# B&R Automation Studio project 2SegDemo (part 2)

#### Cyclic.st
```iecst
PROGRAM _CYCLIC

	FOR i:= 0 TO gMainIf.Cfg.ShuttleCount - 1 DO
		IF NOT gShuttleIf[i].Cmd.Enable AND gShuttleIf[i].Sts.Active THEN
			shState[i] := SH_RESET;
		END_IF

		CASE shState[i] OF
			SH_OFF:  //******************************************************************************** Shuttle is in the off/idle state
				IF gShuttleIf[i].Cmd.Enable THEN
					shState[i] := SH_INIT;
				ELSE

				END_IF
			SH_INIT:  //******************************************************************************** Shuttle is in the initilization state
				//In this state we could make any checks on the current shuttle process perhaps in order to aide in recovery?

				shState[i] := SH_STARTUP;
			SH_STARTUP:  //******************************************************************************** Shuttle is in the startup state
				//In this state maybe we have triggered recovery and we're waiting for the autodrive to complete
				shState[i] := SH_IDLE;

			SH_IDLE:  //************************* ******************************************************* Shuttle is in the idle state
				shFbs[i].MovePlane.Controller := ADR(gMcAcp6DController);
				shFbs[i].MovePlane.ShuttleID := gShuttleIf[i].Cfg.ShuttleId;
				shFbs[i].MovePlane.Velocity := gProcessRecipe.General.Velocity;
				shFbs[i].MovePlane.Acceleration := gProcessRecipe.General.Accel;
				shFbs[i].MovePlane.EndVelocity := 0;
				shFbs[i].MovePlane.PositionX := gLoadStIf.Cfg.StationPos.X;
				shFbs[i].MovePlane.PositionY := gLoadStIf.Cfg.StationPos.Y;
				shFbs[i].MovePlane.Mode := mcACP6D_MOVE_ABSOLUTE;
				shFbs[i].MovePlane.Path := mcACP6D_PATH_Y_THEN_X;
				shFbs[i].MovePlane.Execute := TRUE;

				gShuttleIf[i].Sts.Active := TRUE;
				gShuttleIf[i].Sts.CurrentDestination := DEST_LOAD;

				shState[i] := SH_GO_TO_LOAD;

			SH_GO_TO_LOAD: //******************************************************************************** Shuttle is moving to the load station
				IF shFbs[i].MovePlane.Error THEN
					gShuttleIf[i].Sts.Error := TRUE;
					gShuttleIf[i].Sts.ErrorState := shState[i];

					logArgs[0] := ADR(i);
					logArgs[1] := ADR(shFbs[i].MovePlane.ErrorID);
					logError('ShCtrl','Sh%d had error %d moving to load',ADR(logArgs));

					shState[i] := SH_ERROR;
				ELSIF shFbs[i].MovePlane.Done AND (gLoadStIf.Par.ShuttleIdx = STATION_IS_EMPTY AND gLoadStIf.Sts.ReadyForNewShuttle)
					AND PositionValidation(ADR(gLoadStIf.Cfg.StationPos),ADR(gShuttleIf[i].Sts.ShuttleInfo.Position)) THEN
					gLoadStIf.Par.ShuttleIdx := i;
					gLoadStIf.Cmd.Process := TRUE;

					logArgs[0] := ADR(i);
					logDebug('ShCtrl','Sh%d arrived at Load',ADR(logArgs));

					shFbs[i].MovePlane.Execute := FALSE;
					shState[i] := SH_LOADING;
				END_IF
			SH_LOADING://******************************************************************************** Shuttle is at the load station
				IF gShuttleIf[i].Cmd.NextStep THEN
					gShuttleIf[i].Cmd.NextStep := FALSE;
					gLoadStIf.Cmd.Process := FALSE;

					gShuttleIf[i].Sts.LoopCounter := RandValueDINT(1,gProcessRecipe.General.St1St2Cycles);

					logArgs[0] := ADR(i);
					logDebug('ShCtrl','Sh%d Load complete',ADR(logArgs));

					shState[i] := SH_CHECK_RECIPE;
				END_IF
			SH_CHECK_RECIPE: //******************************************************************************** Shuttle is being checked for the recipe values
				IF gShuttleIf[i].Sts.LoopCounter <= 0 THEN
					shFbs[i].MovePlane.Controller := ADR(gMcAcp6DController);
					shFbs[i].MovePlane.ShuttleID := gShuttleIf[i].Cfg.ShuttleId;
					shFbs[i].MovePlane.Velocity := gProcessRecipe.General.Velocity;
					shFbs[i].MovePlane.Acceleration := gProcessRecipe.General.Accel;
					shFbs[i].MovePlane.EndVelocity := 0;

					shFbs[i].MovePlane.PositionX := gInspectIf.Cfg.StationPos.X;
					shFbs[i].MovePlane.PositionY := gInspectIf.Cfg.StationPos.Y;
					shFbs[i].MovePlane.Mode := mcACP6D_MOVE_ABSOLUTE;
					shFbs[i].MovePlane.Path := mcACP6D_PATH_X_THEN_Y;
					shFbs[i].MovePlane.Execute := TRUE;

					logArgs[0] := ADR(i);
					logDebug('ShCtrl','Sh%d sending to Inspect',ADR(logArgs));

					gShuttleIf[i].Sts.CurrentDestination := DEST_INSPECT;
					shState[i] := SH_GO_TO_INSPECT;
				ELSE

					shFbs[i].MovePlane.Controller := ADR(gMcAcp6DController);
					shFbs[i].MovePlane.ShuttleID := gShuttleIf[i].Cfg.ShuttleId;
					shFbs[i].MovePlane.Velocity := gProcessRecipe.General.Velocity;
					shFbs[i].MovePlane.Acceleration := gProcessRecipe.General.Accel;
					shFbs[i].MovePlane.EndVelocity := 0;

					shFbs[i].MovePlane.Mode := mcACP6D_MOVE_ABSOLUTE;
					shFbs[i].MovePlane.Path := mcACP6D_PATH_Y_THEN_X;
					shFbs[i].MovePlane.Execute := TRUE;

					logArgs[0] := ADR(i);
					logDebug('ShCtrl','Sh%d sending to Station 1',ADR(logArgs));

					gShuttleIf[i].Sts.CurrentDestination := DEST_PROCESS_1;
					shState[i] := SH_GO_TO_ST_1;
				END_IF

			SH_GO_TO_ST_1: //******************************************************************************** Shuttle is going to the #1 operating station
				IF shFbs[i].MovePlane.Error THEN
					gShuttleIf[i].Sts.Error := TRUE;
					gShuttleIf[i].Sts.ErrorState := shState[i];

					logArgs[0] := ADR(i);
					logArgs[1] := ADR(shFbs[i].MovePlane.ErrorID);
					logError('ShCtrl','Sh%d had error %d moving to Station 1',ADR(logArgs));

					shState[i] := SH_ERROR;
				ELSIF shFbs[i].MovePlane.Done AND (gProcessStIf[STATION_1].Par.ShuttleIdx = STATION_IS_EMPTY AND gProcessStIf[STATION_1].Sts.ReadyForNewShuttle)
					AND PositionValidation(ADR(gProcessStIf[STATION_1].Cfg.StationPos),ADR(gShuttleIf[i].Sts.ShuttleInfo.Position)) THEN
					gProcessStIf[STATION_1].Par.ShuttleIdx := i;
					gProcessStIf[STATION_1].Cmd.Process := TRUE;

					logArgs[0] := ADR(i);
					logDebug('ShCtrl','Sh%d arrived at Station 1',ADR(logArgs));

					shFbs[i].MovePlane.Execute := FALSE;
					shState[i] := SH_PREFORM_ST_1;
				END_IF
			SH_PREFORM_ST_1: //******************************************************************************** Shuttle is being operated on at station 1
				IF gShuttleIf[i].Cmd.NextStep THEN
					gShuttleIf[i].Cmd.NextStep := FALSE;

					shFbs[i].MovePlane.Controller := ADR(gMcAcp6DController);
					shFbs[i].MovePlane.ShuttleID := gShuttleIf[i].Cfg.ShuttleId;
					shFbs[i].MovePlane.Velocity := gProcessRecipe.General.Velocity;
					shFbs[i].MovePlane.Acceleration := gProcessRecipe.General.Accel;
					shFbs[i].MovePlane.EndVelocity := 0;
					shFbs[i].MovePlane.PositionX := gProcessStIf[STATION_2].Cfg.StationPos.X;
					shFbs[i].MovePlane.PositionY := gProcessStIf[STATION_2].Cfg.StationPos.Y;
					shFbs[i].MovePlane.Mode := mcACP6D_MOVE_ABSOLUTE;
					shFbs[i].MovePlane.Path := mcACP6D_PATH_Y_THEN_X;
					shFbs[i].MovePlane.Execute := TRUE;

					logArgs[0] := ADR(i);
					logDebug('ShCtrl','Sh%d sent to Station 2',ADR(logArgs));

					gShuttleIf[i].Sts.CurrentDestination := DEST_PROCESS_2;
					shState[i] := SH_GO_TO_ST_2;
				END_IF
			SH_GO_TO_ST_2: //******************************************************************************** Shuttle is going to the #2 operating station
				IF shFbs[i].MovePlane.Error THEN
					gShuttleIf[i].Sts.Error := TRUE;
					gShuttleIf[i].Sts.ErrorState := shState[i];

					logArgs[0] := ADR(i);
					logArgs[1] := ADR(shFbs[i].MovePlane.ErrorID);
					logError('ShCtrl','Sh%d had error %d moving to Station 2',ADR(logArgs));

					shState[i] := SH_ERROR;
				ELSIF shFbs[i].MovePlane.Done AND (gProcessStIf[STATION_2].Par.ShuttleIdx = STATION_IS_EMPTY AND gProcessStIf[STATION_2].Sts.ReadyForNewShuttle)
					AND PositionValidation(ADR(gProcessStIf[STATION_2].Cfg.StationPos),ADR(gShuttleIf[i].Sts.ShuttleInfo.Position)) THEN
					gProcessStIf[STATION_2].Par.ShuttleIdx := i;
					gProcessStIf[STATION_2].Cmd.Process := TRUE;

					logArgs[0] := ADR(i);
					logDebug('ShCtrl','Sh%d arrived at Station 2',ADR(logArgs));

					shFbs[i].MovePlane.Execute := FALSE;
					shState[i] := SH_PREFORM_ST_2;
				END_IF
			SH_PREFORM_ST_2: //******************************************************************************** Shuttle is being operated on at station 2
				IF gShuttleIf[i].Cmd.NextStep THEN
					gShuttleIf[i].Cmd.NextStep := FALSE;

					logArgs[0] := ADR(i);
					logDebug('ShCtrl','Sh%d sent to inspection',ADR(logArgs));

					shState[i] := SH_CHECK_RECIPE;
				END_IF
			SH_GO_TO_INSPECT: //******************************************************************************** Shuttle is going to the inspection station
				IF shFbs[i].MovePlane.Error THEN
					gShuttleIf[i].Sts.Error := TRUE;
					gShuttleIf[i].Sts.ErrorState := shState[i];

					logArgs[0] := ADR(i);
					logArgs[1] := ADR(shFbs[i].MovePlane.ErrorID);
					logError('ShCtrl','Sh%d had error %d moving to inspection',ADR(logArgs));

					shState[i] := SH_ERROR;
				ELSIF shFbs[i].MovePlane.Done AND (gInspectIf.Par.ShuttleIdx = STATION_IS_EMPTY AND gInspectIf.Sts.ReadyForNewShuttle)
						AND PositionValidation(ADR(gInspectIf.Cfg.StationPos),ADR(gShuttleIf[i].Sts.ShuttleInfo.Position)) THEN
					gInspectIf.Par.ShuttleIdx := i;
					gInspectIf.Cmd.Process := TRUE;

					logArgs[0] := ADR(i);
					logDebug('ShCtrl','Sh%d arrived at inspection',ADR(logArgs));

					shFbs[i].MovePlane.Execute := FALSE;
					shState[i] := SH_INSPECT;
				END_IF
			SH_INSPECT: //******************************************************************************** Shuttle is being operated on at the inspection station
				IF gShuttleIf[i].Cmd.NextStep THEN
					gShuttleIf[i].Cmd.NextStep := FALSE;

					shFbs[i].MovePlane.Controller := ADR(gMcAcp6DController);
					shFbs[i].MovePlane.ShuttleID := gShuttleIf[i].Cfg.ShuttleId;
					shFbs[i].MovePlane.Velocity := gProcessRecipe.General.Velocity;
					shFbs[i].MovePlane.Acceleration := gProcessRecipe.General.Accel;
					shFbs[i].MovePlane.EndVelocity := 0;
					shFbs[i].MovePlane.PositionX := gUnloadStIf.Cfg.StationPos.X;
					shFbs[i].MovePlane.PositionY := gUnloadStIf.Cfg.StationPos.Y;
					shFbs[i].MovePlane.Mode := mcACP6D_MOVE_ABSOLUTE;
					shFbs[i].MovePlane.Path := mcACP6D_PATH_Y_THEN_X;
					shFbs[i].MovePlane.Execute := TRUE;

					logArgs[0] := ADR(i);
					logDebug('ShCtrl','Sh%d sent to unload',ADR(logArgs));

					gShuttleIf[i].Sts.CurrentDestination := DEST_UNLOAD;
					shState[i] := SH_GO_TO_UNLOAD;
				END_IF
			SH_GO_TO_UNLOAD: //******************************************************************************** Shuttle is going to the unload station
				IF shFbs[i].MovePlane.Error THEN
					gShuttleIf[i].Sts.Error := TRUE;
					gShuttleIf[i].Sts.ErrorState := shState[i];

					logArgs[0] := ADR(i);
					logArgs[1] := ADR(shFbs[i].MovePlane.ErrorID);
					logError('ShCtrl','Sh%d had error %d moving to unload',ADR(logArgs));

					shState[i] := SH_ERROR;
				ELSIF shFbs[i].MovePlane.Done AND (gUnloadStIf.Par.ShuttleIdx = STATION_IS_EMPTY AND gUnloadStIf.Sts.ReadyForNewShuttle)
						AND PositionValidation(ADR(gUnloadStIf.Cfg.StationPos),ADR(gShuttleIf[i].Sts.ShuttleInfo.Position)) THEN
					gUnloadStIf.Par.ShuttleIdx := i;
					gUnloadStIf.Cmd.Process := TRUE;

					logArgs[0] := ADR(i);
					logDebug('ShCtrl','Sh%d arrived at unload',ADR(logArgs));

					shFbs[i].MovePlane.Execute := FALSE;
					shState[i] := SH_UNLOAD;
				END_IF
			SH_UNLOAD: //******************************************************************************** Shuttle is being operated on at the unload station
				IF gShuttleIf[i].Cmd.NextStep THEN
					gShuttleIf[i].Cmd.NextStep := FALSE;

					shFbs[i].MovePlane.Controller := ADR(gMcAcp6DController);
					shFbs[i].MovePlane.ShuttleID := gShuttleIf[i].Cfg.ShuttleId;
					//shFbs[i].MovePlane.Velocity := gProcessRecipe.General.Velocity;
					shFbs[i].MovePlane.Velocity := 0.5;
					shFbs[i].MovePlane.Acceleration := gProcessRecipe.General.Accel;
					shFbs[i].MovePlane.EndVelocity := 0;
					shFbs[i].MovePlane.PositionX := gLoadStIf.Cfg.StationPos.X;
					shFbs[i].MovePlane.PositionY := gLoadStIf.Cfg.StationPos.Y;
					shFbs[i].MovePlane.Mode := mcACP6D_MOVE_ABSOLUTE;
					shFbs[i].MovePlane.Path := mcACP6D_PATH_Y_THEN_X;
					shFbs[i].MovePlane.Execute := TRUE;

					logArgs[0] := ADR(i);
					logDebug('ShCtrl','Sh%d sent to load',ADR(logArgs));
					gShuttleIf[i].Cmd.ResetProductInfo := TRUE;

					gShuttleIf[i].Sts.CurrentDestination := DEST_LOAD;
					shState[i] := SH_GO_TO_LOAD;
				END_IF
			SH_STOPPING: //******************************************************************************** Shuttle is in the stopping state
				IF shFbs[i].Stop.Error THEN
					shState[i] := SH_ERROR;
				ELSIF gShuttleIf[i].Sts.ShuttleInfo.State.Valid AND
						(gShuttleIf[i].Sts.ShuttleInfo.State.Value = mcACP6D_SH_STATE_IDLING OR gShuttleIf[i].Sts.ShuttleInfo.State.Value = mcACP6D_SH_STATE_DISABLED) THEN
					gShuttleIf[i].Cmd.NextStep := FALSE;

					shFbs[i].Stop.Execute := FALSE;
					shFbs[i].MovePlane.Execute := FALSE;
					shFbs[i].ShRunMacroFb.Execute := FALSE;

					shState[i] := SH_RESET;
				END_IF

			SH_ERROR: //******************************************************************************** Shuttle is in the error state
				IF gShuttleIf[i].Cmd.Reset THEN
					shState[i] := SH_RESET;
				END_IF
			SH_RESET: //******************************************************************************** Reset all shuttle values
				gShuttleIf[i].Cmd.ResetProductInfo := TRUE;
				gShuttleIf[i].Cmd.Reset := FALSE;
				gShuttleIf[i].Cmd.NextStep := FALSE;
				gShuttleIf[i].Cmd.RunProcessDemo := FALSE;

				gShuttleIf[i].Sts.Active := FALSE;

				shFbs[i].MovePlane.Execute := FALSE;
				shFbs[i].ShRunMacroFb.Execute := FALSE;
				shFbs[i].Stop.Execute := FALSE;

				shState[i] := SH_OFF;
		END_CASE;

		shFbs[i].Stop();
		shFbs[i].MovePlane();

		IF gShuttleIf[i].Cmd.ResetProductInfo THEN
			gShuttleIf[i].Sts.Error := FALSE;
			gShuttleIf[i].Sts.ErrorState := 0;
			gShuttleIf[i].Cmd.ResetProductInfo := FALSE;
			gShuttleIf[i].Sts.LoopCounter := 0;
			gShuttleIf[i].Sts.ProductState := PROD_EMPTY;
			brsmemset(ADR(gShuttleIf[i].Sts.ProdFill),0,SIZEOF(gShuttleIf[i].Sts.ProdFill));
		END_IF

	END_FOR;

	pDebugIf ACCESS ADR(gShuttleIf[debugIdx]);
	pDebugState ACCESS ADR(shState[debugIdx]);
	pDebugFbs ACCESS ADR(shFbs[debugIdx]);

END_PROGRAM
```

#### Init.st
```iecst
PROGRAM _INIT

	FOR i:=0 TO gMainIf.Cfg.ShuttleCount-1 DO
		gShuttleIf[i].Par.X := 0.06;
		gShuttleIf[i].Par.Y := 0.06 * (i + 1) + 0.06*i;
		gShuttleIf[i].Par.Accel := 10;
		gShuttleIf[i].Par.Vel := 0.5;
		gShuttleIf[i].Par.EndVel := 0;
	END_FOR;
	gProcessRecipe.General.Velocity := 1;
	gProcessRecipe.General.Accel := 10;
END_PROGRAM
```

### Program Logical/Source/ShuttleCtrl/Recovery (IEC)

#### Types.typ
```iecst
TYPE
	RecoveryFbs : 	STRUCT
		AsyncMoveFb : MC_BR_MoveInPlaneAsync_Acp6D;
		ShStopFb : MC_BR_Stop_Acp6D;
		DelayFb : TON;
	END_STRUCT;
	RecoveryStateEnum :
		(
		RECOVER_IDLE, (*Recovery is in an idle state*)
		RECOVER_INIT, (*Initalize recovery state*)
		RECOVER_AUTODRIVE, (*Preform autodrive movement for recovery*)
		RECOVER_STOP,
		RECOVER_DONE, (*Recovery has been completed*)
		RECOVER_ERROR (*Recovery had an error*)
		);
END_TYPE
```

#### Variables.var
```iecst
VAR
	state : RecoveryStateEnum;
	RecoverFbs : RecoveryFbs;
	i : USINT;
END_VAR
```

#### Cyclic.st
```iecst
PROGRAM _CYCLIC

	(*
	Shuttle reocvery
		Move all shuttles to autodrive positions
		Wait for autodrive to be finished
		loop through each shuttle
			if that shuttle's group is current
				it is not recovered,
					groupRecovered=false
					Evaluate each shuttle's position
					Send it to the unload position and set the "Next step cmd" to be true
				else
					onwards, do nothing

	*)

	CASE state OF
		RECOVER_IDLE:   //******************************************************************************** Recovery is in an idle state*)
			IF g6DRecoveryIf.Cmd.Recover THEN
				g6DRecoveryIf.Sts.Recovering := TRUE;
				state := RECOVER_INIT;
			END_IF
		RECOVER_INIT:   //******************************************************************************** Initalize recovery state*)
			RecoverFbs.AsyncMoveFb.Controller := ADR(gMcAcp6DController);
			RecoverFbs.AsyncMoveFb.NumberOfShuttles := gMainIf.Cfg.ShuttleCount;
			RecoverFbs.AsyncMoveFb.Velocity := g6DRecoveryIf.Par.Vel;
			RecoverFbs.AsyncMoveFb.Acceleration := g6DRecoveryIf.Par.Accel;
			FOR i:=0 TO gMainIf.Cfg.ShuttleCount - 1 DO
				RecoverFbs.AsyncMoveFb.PositionX[i] := g6DRecoveryIf.Par.AutoDrivePositions[i].X;
				RecoverFbs.AsyncMoveFb.PositionY[i] := g6DRecoveryIf.Par.AutoDrivePositions[i].Y;
				RecoverFbs.AsyncMoveFb.ShuttleID[i] := gShuttleIf[g6DRecoveryIf.Par.AutoDrivePositions[i].ShIdx].Cfg.ShuttleId;
				IF RecoverFbs.AsyncMoveFb.ShuttleID[i] = 0 THEN// Invalid shuttle id here
					g6DRecoveryIf.Sts.Error := TRUE;
				END_IF
			END_FOR;
			IF NOT g6DRecoveryIf.Sts.Error THEN
				RecoverFbs.AsyncMoveFb.Execute := TRUE;
				state := RECOVER_AUTODRIVE;
			ELSE
				state := RECOVER_ERROR;
			END_IF

		RECOVER_AUTODRIVE:   //******************************************************************************** Preform autodrive movement for recovery*)
			IF RecoverFbs.AsyncMoveFb.Error AND RecoverFbs.AsyncMoveFb.ErrorID = mcACP6D_ERR_WRONG_SH_STATE THEN
				RecoverFbs.AsyncMoveFb.Execute := FALSE;

				RecoverFbs.DelayFb.IN := TRUE;
				RecoverFbs.DelayFb.PT := T#5s;

				RecoverFbs.ShStopFb.Controller := ADR(gMcAcp6DController);
				RecoverFbs.ShStopFb.ShuttleID := 0;
				RecoverFbs.ShStopFb.Execute := TRUE;

				state := RECOVER_STOP;
			ELSIF RecoverFbs.AsyncMoveFb.Error THEN
				g6DRecoveryIf.Sts.Error := TRUE;
				state := RECOVER_ERROR;
			ELSIF RecoverFbs.AsyncMoveFb.Done THEN
				g6DRecoveryIf.Sts.ReadyToStartProc := TRUE;
				RecoverFbs.AsyncMoveFb.Execute := FALSE;

				state := RECOVER_DONE;
			END_IF
		RECOVER_STOP:  //******************************************************************************** Stop All shuttles
			IF RecoverFbs.ShStopFb.Error THEN
				g6DRecoveryIf.Sts.Error := TRUE;
				state := RECOVER_ERROR;
			ELSIF RecoverFbs.ShStopFb.Done AND RecoverFbs.DelayFb.Q THEN
				RecoverFbs.DelayFb.IN := FALSE;
				RecoverFbs.ShStopFb.Execute := FALSE;

				RecoverFbs.AsyncMoveFb.Execute := TRUE;

				state := RECOVER_AUTODRIVE;
			END_IF
		RECOVER_DONE:   //******************************************************************************** Recovery has been completed*)
			IF NOT g6DRecoveryIf.Cmd.Recover THEN
				g6DRecoveryIf.Cmd.Reset := FALSE;
				RecoverFbs.DelayFb.IN := FALSE;
				g6DRecoveryIf.Sts.Done := FALSE;
				g6DRecoveryIf.Sts.ReadyToStartProc := FALSE;
				g6DRecoveryIf.Sts.Recovering := FALSE;
				g6DRecoveryIf.Sts.ShuttlesRecovered := FALSE;
				g6DRecoveryIf.Sts.Error := FALSE;

				RecoverFbs.AsyncMoveFb.Execute := FALSE;
				state := RECOVER_IDLE;
			END_IF
		RECOVER_ERROR:   //******************************************************************************** Recovery had an error*)
			IF g6DRecoveryIf.Cmd.Reset THEN
				RecoverFbs.DelayFb.IN := FALSE;
				g6DRecoveryIf.Cmd.Reset := FALSE;
				g6DRecoveryIf.Cmd.Recover := FALSE;

				g6DRecoveryIf.Sts.Done := FALSE;
				g6DRecoveryIf.Sts.ReadyToStartProc := FALSE;
				g6DRecoveryIf.Sts.Recovering := FALSE;
				g6DRecoveryIf.Sts.ShuttlesRecovered := FALSE;
				g6DRecoveryIf.Sts.Error := FALSE;

				RecoverFbs.AsyncMoveFb.Execute := FALSE;
				RecoverFbs.ShStopFb.Execute := FALSE;
				state := RECOVER_IDLE;
			END_IF
	END_CASE;
	RecoverFbs.AsyncMoveFb();
	RecoverFbs.ShStopFb();
	RecoverFbs.DelayFb();
END_PROGRAM
```

#### Init.st
```iecst
PROGRAM _INIT
	g6DRecoveryIf.Par.Vel := 1;
	g6DRecoveryIf.Par.Accel := 10;

	//************************************************************************* Shuttle 1
	g6DRecoveryIf.Par.AutoDrivePositions[0].ShIdx := 0;
	g6DRecoveryIf.Par.AutoDrivePositions[0].X := 0.42;
	g6DRecoveryIf.Par.AutoDrivePositions[0].Y := 0.18;
	//************************************************************************* Shuttle 2
	g6DRecoveryIf.Par.AutoDrivePositions[1].ShIdx := 1;
	g6DRecoveryIf.Par.AutoDrivePositions[1].X := 0.30;
	g6DRecoveryIf.Par.AutoDrivePositions[1].Y := 0.18;
	//************************************************************************* Shuttle 3
	g6DRecoveryIf.Par.AutoDrivePositions[2].ShIdx := 2;
	g6DRecoveryIf.Par.AutoDrivePositions[2].X := 0.42;
	g6DRecoveryIf.Par.AutoDrivePositions[2].Y := 0.30;
	//************************************************************************* Shuttle 4
	g6DRecoveryIf.Par.AutoDrivePositions[3].ShIdx := 3;
	g6DRecoveryIf.Par.AutoDrivePositions[3].X := 0.30;
	g6DRecoveryIf.Par.AutoDrivePositions[3].Y := 0.30;
	//************************************************************************* Shuttle 5
	g6DRecoveryIf.Par.AutoDrivePositions[4].ShIdx := 4;
	g6DRecoveryIf.Par.AutoDrivePositions[4].X := 0.42;
	g6DRecoveryIf.Par.AutoDrivePositions[4].Y := 0.42;
	//************************************************************************* Shuttle 6
	g6DRecoveryIf.Par.AutoDrivePositions[5].ShIdx := 5;
	g6DRecoveryIf.Par.AutoDrivePositions[5].X := 0.30;
	g6DRecoveryIf.Par.AutoDrivePositions[5].Y := 0.42;
	//************************************************************************* Shuttle 7
	g6DRecoveryIf.Par.AutoDrivePositions[6].ShIdx := 6;
	g6DRecoveryIf.Par.AutoDrivePositions[6].X := 0.42;
	g6DRecoveryIf.Par.AutoDrivePositions[6].Y := 0.54;
	//************************************************************************* Shuttle 8
	g6DRecoveryIf.Par.AutoDrivePositions[7].ShIdx := 7;
	g6DRecoveryIf.Par.AutoDrivePositions[7].X := 0.30;
	g6DRecoveryIf.Par.AutoDrivePositions[7].Y := 0.54;

END_PROGRAM
```

### Program Logical/Source/ShuttleCtrl/ProcessDemoCtrl (IEC) - Control the process demo

#### Types.typ
```iecst
TYPE
	ProcessDemoStateEnum :
		(
		PROCESS_IDLE,
		PROCESS_ROUTING,
		PROCESS_STARTUP,
		PROCESS_RUN_DEMO,
		PROCESS_STOPPING_STATIONS,
		PROCESS_STOPPING,
		PROCESS_UNLOAD_PROGRAM,
		PROCESS_ERROR,
		PROCESS_RESET
		);
	ProcessDemoFbsTyp : 	STRUCT
		Stop6DFb : MC_BR_Stop_Acp6D;
		MoveProgramFb : MC_BR_MoveProgram;
		StopRobotFb : MC_GroupStop;
		UnloadProgramFb : MC_BR_UnloadProgram;
	END_STRUCT;
END_TYPE
```

#### Variables.var
```iecst
VAR
	state : ProcessDemoStateEnum;
	Fbs : ProcessDemoFbsTyp;
	i : USINT;
END_VAR
```

#### Cyclic.st
```iecst
(* This task control the demo routine for the process demo
	The robot and the 6D are expected to be powered on, homed and not in any error states before starting this demo

	Recovery
	Robot Setup
	Enable Stations
	Run Demo
	Error
	Stopping
	Reset
*)

PROGRAM _CYCLIC
	CASE state OF
		PROCESS_IDLE:  //******************************************************************************** Idle Wait State
			IF gProcessPickPlaceIf.Cmd.RunDemo THEN
				g6DRecoveryIf.Cmd.Recover := TRUE;

				state := PROCESS_ROUTING;
			ELSIF gProcessPickPlaceIf.Cmd.Reset THEN
				state := PROCESS_RESET;
			END_IF
		PROCESS_ROUTING:  //******************************************************************************** Running the routing demo
			IF g6DRecoveryIf.Sts.Error THEN
				gProcessPickPlaceIf.Sts.Error := TRUE;
				state := PROCESS_ERROR;
			ELSIF (g6DRecoveryIf.Sts.ReadyToStartProc) THEN
				g6DRecoveryIf.Cmd.Recover := FALSE;

				gLoadStIf.Cmd.Enable := TRUE;
				//gUnloadStIf.Cmd.Enable := TRUE; The Load station will enable the Unload station in order to complete the Load process first
				gProcessStIf[STATION_1].Cmd.Enable := TRUE;
				gProcessStIf[STATION_2].Cmd.Enable := TRUE;
				gInspectIf.Cmd.Enable := TRUE;

				Fbs.MoveProgramFb.AxesGroup := ADR(g3AxDeltaA);
				Fbs.MoveProgramFb.Name := 'ProcessDemo.gcode';
				Fbs.MoveProgramFb.Execute := TRUE;

				state := PROCESS_STARTUP;
			END_IF
		PROCESS_STARTUP:  //******************************************************************************** Starting up the demos state
			IF gLoadStIf.Sts.Error OR
					gInspectIf.Sts.Error OR
					gProcessStIf[STATION_1].Sts.Error OR
					gProcessStIf[STATION_2].Sts.Error OR
					Fbs.MoveProgramFb.Error THEN
				gProcessPickPlaceIf.Sts.Error := TRUE;
				state := PROCESS_ERROR;
			ELSIF (gLoadStIf.Sts.Enabled AND
					//gUnloadStIf.Sts.Enabled AND The load station enables the unload station once the startup process has completed
					gInspectIf.Cmd.Enable AND
					gProcessStIf[STATION_1].Sts.Enabled AND
					gProcessStIf[STATION_2].Sts.Enabled OR NOT gMainIf.Cfg.Enable6D)
					AND
					Fbs.MoveProgramFb.Phase = mcPRGPH_REAL_RUN THEN

				CmdShEnable(TRUE, ADR(gShuttleIf),gMainIf.Cfg.ShuttleCount);

				gProcessPickPlaceIf.Sts.DemoRunning := TRUE;

				state := PROCESS_RUN_DEMO;

			END_IF
		PROCESS_RUN_DEMO:  //******************************************************************************** Running the process demo
			IF Fbs.MoveProgramFb.Error OR
					gLoadStIf.Sts.Error OR
					gUnloadStIf.Sts.Error OR
					gProcessStIf[STATION_1].Sts.Error OR
					gProcessStIf[STATION_2].Sts.Error OR
					gInspectIf.Sts.Error THEN
				state := PROCESS_ERROR;
			ELSIF NOT gProcessPickPlaceIf.Cmd.RunDemo THEN
				gLoadStIf.Cmd.Enable := FALSE;
				gUnloadStIf.Cmd.Enable := FALSE;
				gProcessStIf[STATION_1].Cmd.Enable := FALSE;
				gProcessStIf[STATION_2].Cmd.Enable := FALSE;
				gInspectIf.Cmd.Enable := FALSE;

				state := PROCESS_STOPPING_STATIONS;
			END_IF
		PROCESS_STOPPING_STATIONS:  //******************************************************************************** Stopping the Stations
			gLoadStIf.Cmd.Enable := FALSE;
			gUnloadStIf.Cmd.Enable := FALSE;
			gProcessStIf[STATION_1].Cmd.Enable := FALSE;
			gProcessStIf[STATION_2].Cmd.Enable := FALSE;
			gInspectIf.Cmd.Enable := FALSE;
			IF (NOT gLoadStIf.Sts.Enabled AND
					//gUnloadStIf.Sts.Enabled AND The load station enables the unload station once the startup process has completed
					NOT gInspectIf.Cmd.Enable AND
					NOT gProcessStIf[STATION_1].Sts.Enabled AND
					NOT gProcessStIf[STATION_2].Sts.Enabled AND NOT gUnloadStIf.Sts.Enabled) AND Fbs.MoveProgramFb.Done
					THEN

				Fbs.StopRobotFb.AxesGroup := ADR(g3AxDeltaA);
				Fbs.StopRobotFb.Execute := TRUE;

				Fbs.Stop6DFb.Controller := ADR(gMcAcp6DController);
				Fbs.Stop6DFb.ShuttleID := 0;
				Fbs.Stop6DFb.Execute := TRUE;

				state := PROCESS_STOPPING;
			END_IF
		PROCESS_STOPPING:  //******************************************************************************** Stopping the demo
			IF Fbs.Stop6DFb.Error OR Fbs.StopRobotFb.Error THEN
				gProcessPickPlaceIf.Sts.Error := TRUE;

				state := PROCESS_ERROR;
			ELSIF Fbs.Stop6DFb.Done AND Fbs.StopRobotFb.Done THEN
				Fbs.StopRobotFb.Execute := FALSE;
				Fbs.Stop6DFb.Execute := FALSE;

				gProcessPickPlaceIf.Sts.DemoRunning := FALSE;

				FOR i:=0 TO gMainIf.Cfg.ShuttleCount - 1 DO
					gShuttleIf[i].Cmd.Enable := FALSE;
					gShuttleIf[i].Sts.Recovered := FALSE;
				END_FOR;

				Fbs.UnloadProgramFb.AxesGroup := ADR(g3AxDeltaA);
				Fbs.UnloadProgramFb.Execute := TRUE;
				Fbs.UnloadProgramFb.Mode := mcUNLOADPRG_ALL;

				state := PROCESS_UNLOAD_PROGRAM;
			END_IF
		PROCESS_UNLOAD_PROGRAM:   //******************************************************************************** Unloading the program
			IF Fbs.UnloadProgramFb.Error THEN
				gProcessPickPlaceIf.Sts.Error := TRUE;

				state := PROCESS_ERROR;
			ELSIF Fbs.UnloadProgramFb.Done THEN
				Fbs.UnloadProgramFb.Execute := FALSE;

				state := PROCESS_RESET;
			END_IF

		PROCESS_ERROR:  //******************************************************************************** Demo in error state
			IF gProcessPickPlaceIf.Cmd.Reset THEN
				gLoadStIf.Cmd.Reset := TRUE;
				gUnloadStIf.Cmd.Reset:= TRUE;
				gProcessStIf[STATION_1].Cmd.Reset := TRUE;
				gProcessStIf[STATION_2].Cmd.Reset := TRUE;
				gInspectIf.Cmd.Reset := TRUE;

				Fbs.Stop6DFb.Controller := ADR(gMcAcp6DController);
				Fbs.Stop6DFb.ShuttleID := 0;
				Fbs.Stop6DFb.Execute := TRUE;

				FOR i:= 0 TO gMainIf.Cfg.ShuttleCount - 1 DO
					gShuttleIf[i].Cmd.Enable := FALSE;
					gShuttleIf[i].Cmd.Reset := TRUE;
				END_FOR;
				state := PROCESS_RESET;
			END_IF
		PROCESS_RESET:  //******************************************************************************** Resetting the demo state
			Fbs.Stop6DFb.Execute := FALSE;
			Fbs.MoveProgramFb.Execute := FALSE;
			Fbs.StopRobotFb.Execute := FALSE;
			Fbs.UnloadProgramFb.Execute := FALSE;

			gDelta.Cmd.ErrorReset := gDelta.Status.Error;

			g6DRecoveryIf.Cmd.Reset := g6DRecoveryIf.Sts.Error;

			gLoadStIf.Cmd.Enable := FALSE;
			gUnloadStIf.Cmd.Enable := FALSE;
			gProcessStIf[STATION_1].Cmd.Enable := FALSE;
			gProcessStIf[STATION_2].Cmd.Enable := FALSE;
			gInspectIf.Cmd.Enable := FALSE;

			gProcessPickPlaceIf.Cmd.PickLoad := FALSE;
			gProcessPickPlaceIf.Cmd.PickUnload := FALSE;
			gProcessPickPlaceIf.Cmd.RunDemo := FALSE;
			gProcessPickPlaceIf.Cmd.GetLoadPart := FALSE;

			gProcessPickPlaceIf.Sts.Error := FALSE;
			gProcessPickPlaceIf.Sts.DemoRunning := FALSE;
			gProcessPickPlaceIf.Sts.FinishedProductPresent := FALSE;
			gProcessPickPlaceIf.Sts.ReadyForLoad := FALSE;
			gProcessPickPlaceIf.Sts.ReadyForUnload := FALSE;
			gProcessPickPlaceIf.Sts.StartupComplete := FALSE;
			gProcessPickPlaceIf.Sts.Sync := FALSE;
			gProcessPickPlaceIf.Sts.UnfinishedProductPresent := FALSE;
			gProcessPickPlaceIf.Cmd.Reset := FALSE;
			gProcessPickPlaceIf.Sts.Place := FALSE;

			state := PROCESS_IDLE;
	END_CASE;

	Fbs.Stop6DFb();
	Fbs.MoveProgramFb();
	Fbs.UnloadProgramFb();
	Fbs.StopRobotFb();
END_PROGRAM
```

#### Init.st
```iecst
PROGRAM _INIT
	gDanceDemoIf.Par.DemoTime := T#30s;

END_PROGRAM
```

### DemoGlobalVariables.var
```iecst
VAR
	gSyncConoyDemoIf : IndvDanceDemoIfTyp;
	gDofDemoIf : IndvDanceDemoIfTyp;
	gRoutingDemoIf : IndvDanceDemoIfTyp;
END_VAR
```

### DemoGlobalTypes.typ
```iecst
TYPE
	IndvDanceDemoIfTyp : 	STRUCT
		Cmd : IndvDanceDemoCmdTyp;
		Par : IndvDanceDemoParTyp;
		Sts : IndvDanceDemoStsTyp;
	END_STRUCT;
	IndvDanceDemoCmdTyp : 	STRUCT
		Run : BOOL;
		Reset : BOOL;
	END_STRUCT;
	IndvDanceDemoStsTyp : 	STRUCT
		Running : BOOL;
		Error : BOOL;
		Active : BOOL;
	END_STRUCT;
	IndvDanceDemoParTyp : 	STRUCT
		RobotVelocity : REAL;
		RobotProgramName : STRING[260];
	END_STRUCT;
END_TYPE
```

### Program Logical/Source/Demos/WaveDemo (IEC)

#### Types.typ
```iecst
TYPE
	WaveParsTyp : 	STRUCT
		Amp : REAL;
		Center : REAL;
		Freq : REAL;
		X : REAL;
		Y : REAL;
	END_STRUCT;
	ShuttleOutputTyp : 	STRUCT
		Height : REAL;
		Angle : REAL;
		X : REAL;
	END_STRUCT;
	WaveStateEnum :
		(
		WAVE_IDLE,
		WAVE_MOVE_TO_START,
		WAVE_CREATE_GROUP,
		WAVE_BOND_GROUP,
		WAVE_CFG_CHANNEL,
		WAVE_SET_HEIGHT,
		WAVE_WAVE,
		WAVE_EXIT_CFG,
		WAVE_STOP,
		WAVE_MOVE_BACK,
		WAVE_UNBOUND_GROUP,
		WAVE_DELETE_GROUP,
		WAVE_ERROR
		);
	WaveFbsTyp : 	STRUCT
		CyclicChCtrlFb : MC_BR_WriteCyclicChCtrl_Acp6D;
		CyclicZFb : MC_BR_WriteCyclicCh_Acp6D;
		CyclicRxFb : MC_BR_WriteCyclicCh_Acp6D;
		CyclicXFb : MC_BR_WriteCyclicCh_Acp6D;
		AutoDriveFB : MC_BR_MoveInPlaneAsync_Acp6D;
		GroupCreateFb : MC_BR_ShGroupCreate_Acp6D;
		GroupDeleteFb : MC_BR_ShGroupDelete_Acp6D;
		GroupCtrlFb : MC_BR_ShGroupCoupleCtrl_Acp6D;
		ShortAxisFb : MC_BR_MoveShortAxis_Acp6D;
	END_STRUCT;
END_TYPE
```

#### Variables.var
```iecst
VAR
	startRef : ShuttleOutputTyp;
	Wavepars : WaveParsTyp;
	ShCtrl : ShuttleOutputTyp;
	Fbs : WaveFbsTyp;
	state : WaveStateEnum;
	wave : BOOL;
	shId : USINT;
	defaultLevitationHeight : REAL;
	Slide : WaveParsTyp;
	Reset : BOOL;
END_VAR
```

#### Cyclic.st
```iecst
//Hz is times per second, in this case times is revolutions.
//To convert the Hz to revolutions and then scale by the task class cycle time
//1 hz, would mean that every TC cycle, we'd be incrementing by 2*PI/CycleTime

//Rx and Rz cylcic positions are always relative to the current position at the
//  ENABLING of the cyclic channel. Why? Who knows but that's the way it works

PROGRAM _CYCLIC
	Wavepars.X := Wavepars.X + Wavepars.Freq / 1000 * 2 * 3.14;
	Slide.X := Slide.X + Slide.Freq / 1000 * 2 * 3.14;
	IF Wavepars.X > 2 * 3.14 THEN
		Wavepars.X := 0;
	END_IF

	IF Slide.X > 2 * 3.14 THEN
		Slide.X := 0;
	END_IF

	Wavepars.Y := SIN(Wavepars.X);
	ShCtrl.Height := Wavepars.Y * Wavepars.Amp + Wavepars.Center;

	//For the angle,just going to scale between -20/+20mRad.
	ShCtrl.Angle := COS(Wavepars.X) * 20;

	ShCtrl.X := SIN(Slide.X) * 180 + 240;

	CASE state OF
		WAVE_IDLE: //**************************************************************** Idle State
			IF wave THEN
				Fbs.AutoDriveFB.Controller := ADR(gMcAcp6DController);
				Fbs.AutoDriveFB.Velocity := 1.0;
				Fbs.AutoDriveFB.Acceleration := 10.0;
				Fbs.AutoDriveFB.ShuttleID[0] := 1;
				Fbs.AutoDriveFB.ShuttleID[1] := 2;
				Fbs.AutoDriveFB.NumberOfShuttles := 2;
				Fbs.AutoDriveFB.PositionX[0] := 0.420;
				Fbs.AutoDriveFB.PositionX[1] := 0.420;
				Fbs.AutoDriveFB.PositionY[0] := 0.055;
				Fbs.AutoDriveFB.PositionY[1] := 0.185;
				Fbs.AutoDriveFB.Execute := TRUE;

				state := WAVE_MOVE_TO_START;
			END_IF
		WAVE_MOVE_TO_START: //**************************************************************** Move to the start position
			IF Fbs.AutoDriveFB.Error THEN
				state := WAVE_ERROR;
			ELSIF Fbs.AutoDriveFB.Done THEN
				Fbs.AutoDriveFB.Execute := FALSE;

				Fbs.GroupCreateFb.Controller := ADR(gMcAcp6DController);
				Fbs.GroupCreateFb.GroupID := 1;
				Fbs.GroupCreateFb.NumberOfShuttles := 2;
				Fbs.GroupCreateFb.ShuttleID[0] := 1;
				Fbs.GroupCreateFb.ShuttleID[1] := 2;
				Fbs.GroupCreateFb.Execute := TRUE;

				state := WAVE_CREATE_GROUP;
			END_IF
		WAVE_CREATE_GROUP: //**************************************************************** Create Sh Group
			IF Fbs.GroupCreateFb.Error THEN
				state := WAVE_ERROR;
			ELSIF Fbs.GroupCreateFb.Done THEN
				Fbs.GroupCreateFb.Execute := FALSE;

				Fbs.GroupCtrlFb.Controller := ADR(gMcAcp6DController);
				Fbs.GroupCtrlFb.CoupleMode := mcACP6D_GROUP_COUPLE_ONLY_XY;
				Fbs.GroupCtrlFb.GroupID := 1;
				Fbs.GroupCtrlFb.Option := mcACP6D_GROUP_COUPLE;
				Fbs.GroupCtrlFb.Execute := TRUE;

				state := WAVE_BOND_GROUP;
			END_IF
		WAVE_BOND_GROUP: //**************************************************************** Bond Sh Group
			IF Fbs.GroupCtrlFb.Error THEN
				state := WAVE_ERROR;
			ELSIF Fbs.GroupCtrlFb.Done THEN
				Fbs.GroupCtrlFb.Execute := FALSE;

				Fbs.ShortAxisFb.Controller := ADR(gMcAcp6DController);
				Fbs.ShortAxisFb.ShuttleID := shId;
				Fbs.ShortAxisFb.PositionZ := (Wavepars.Amp + Wavepars.Center) / 1000.0;
				Fbs.ShortAxisFb.PositionRx := 0.0;
				Fbs.ShortAxisFb.PositionRy := 0;
				Fbs.ShortAxisFb.PositionRz := 0;
				Fbs.ShortAxisFb.VelocityZ := 1;
				Fbs.ShortAxisFb.VelocityRx := 1;
				Fbs.ShortAxisFb.VelocityRy := 1;
				Fbs.ShortAxisFb.VelocityRz := 1;
				Fbs.ShortAxisFb.Execute := TRUE;

				startRef.Height := Fbs.ShortAxisFb.PositionZ;
				startRef.Angle := Fbs.ShortAxisFb.PositionRx;

				state := WAVE_CFG_CHANNEL;
			END_IF
		WAVE_CFG_CHANNEL: //**************************************************************** Configure cyclic channel
			IF Fbs.ShortAxisFb.Error THEN
				state := WAVE_ERROR;
			ELSIF Fbs.ShortAxisFb.Done THEN
				Fbs.ShortAxisFb.Execute := FALSE;

				//Wavepars.Freq := 1.0;
				Wavepars.X := 1.57;
				Slide.X := 1.57;
				Wavepars.Y := SIN(Wavepars.X);
				ShCtrl.Height := Wavepars.Y * Wavepars.Amp + Wavepars.Center;

				//For the angle,just going to scale between -25/+25mRad.
				ShCtrl.Angle := COS(Wavepars.X) * 25;

				Fbs.CyclicZFb.AxisID := 3;
				Fbs.CyclicZFb.ChannelID := 1;
				Fbs.CyclicZFb.Controller := ADR(gMcAcp6DController);
				Fbs.CyclicZFb.Value := (Wavepars.Amp + Wavepars.Center) - ShCtrl.Height ;
				Fbs.CyclicZFb.Enable := TRUE;

				Fbs.CyclicRxFb.AxisID := 5;
				Fbs.CyclicRxFb.ChannelID := 1;
				Fbs.CyclicRxFb.Controller := ADR(gMcAcp6DController);
				Fbs.CyclicRxFb.Value := 0;
				Fbs.CyclicRxFb.Enable := TRUE;

				Fbs.CyclicXFb.AxisID := 1;
				Fbs.CyclicXFb.ChannelID := 1;
				Fbs.CyclicXFb.Controller := ADR(gMcAcp6DController);
				Fbs.CyclicXFb.Value := 0.42;
				Fbs.CyclicXFb.Enable := TRUE;
				state := WAVE_SET_HEIGHT;
			END_IF

		WAVE_SET_HEIGHT: //**************************************************************** Set the starting height
			Fbs.CyclicChCtrlFb.Controller := ADR(gMcAcp6DController);
			Fbs.CyclicChCtrlFb.ShuttleID[0] := shId;
			Fbs.CyclicChCtrlFb.ChannelID[0] := 1;
			Fbs.CyclicChCtrlFb.AxisID[0].0 := TRUE; //X
			Fbs.CyclicChCtrlFb.AxisID[0].2 := TRUE; //Z
			Fbs.CyclicChCtrlFb.AxisID[0].4 := TRUE; //Ry
			Fbs.CyclicChCtrlFb.Execute := TRUE;
			Fbs.CyclicChCtrlFb.NumberOfShuttles := 1;
			Fbs.CyclicChCtrlFb.Level := 1;

//			Wavepars.Freq := 1.5;
//			Slide.Freq := 0.05;

			IF Fbs.CyclicChCtrlFb.Error THEN
				state := WAVE_ERROR;
			ELSIF Fbs.CyclicChCtrlFb.Done THEN
				Fbs.CyclicChCtrlFb.Execute := FALSE;

				//state := WAVE_WAVE;
				state := WAVE_ERROR;
			END_IF
		WAVE_WAVE: //**************************************************************** Write channels, ride the wave
			Fbs.CyclicZFb.Value := -((Wavepars.Amp + Wavepars.Center) - ShCtrl.Height) / 1000.0;
			Fbs.CyclicRxFb.Value := ShCtrl.Angle / 1000.0;
			Fbs.CyclicXFb.Value := ShCtrl.X / 1000.0;

			IF NOT wave THEN
				Fbs.CyclicZFb.Enable := FALSE;
				Fbs.CyclicRxFb.Enable := FALSE;
				Fbs.CyclicXFb.Enable := FALSE;
				Fbs.CyclicChCtrlFb.Execute := TRUE;
				Fbs.CyclicChCtrlFb.Level := 0;

				state := WAVE_EXIT_CFG;
			END_IF
		WAVE_EXIT_CFG:  //**************************************************************** Exit config channel
			IF Fbs.CyclicChCtrlFb.Error THEN
				state := WAVE_ERROR;
			ELSIF Fbs.CyclicChCtrlFb.Done THEN
				Fbs.CyclicChCtrlFb.Execute := FALSE;

				Fbs.ShortAxisFb.Controller := ADR(gMcAcp6DController);
				Fbs.ShortAxisFb.ShuttleID := shId;
				Fbs.ShortAxisFb.PositionZ := defaultLevitationHeight;
				Fbs.ShortAxisFb.PositionRx := 0.0;
				Fbs.ShortAxisFb.PositionRy := 0;
				Fbs.ShortAxisFb.PositionRz := 0;
				Fbs.ShortAxisFb.VelocityZ := 1;
				Fbs.ShortAxisFb.VelocityRx := 1;
				Fbs.ShortAxisFb.VelocityRy := 1;
				Fbs.ShortAxisFb.VelocityRz := 1;
				Fbs.ShortAxisFb.Execute := TRUE;

				state := WAVE_MOVE_BACK;
			END_IF
		WAVE_MOVE_BACK: //**************************************************************** Move Back to level
			IF Fbs.ShortAxisFb.Error THEN
				state := WAVE_ERROR;
			ELSIF Fbs.ShortAxisFb.Done THEN
				Fbs.ShortAxisFb.Execute := FALSE;

				Fbs.GroupCtrlFb.Option := mcACP6D_GROUP_DECOUPLE;
				Fbs.GroupCtrlFb.Execute := TRUE;

				state := WAVE_UNBOUND_GROUP;
			END_IF
		WAVE_UNBOUND_GROUP: //**************************************************************** Unbond Sh Group
			IF Fbs.GroupCtrlFb.Error THEN
				state := WAVE_ERROR;
			ELSIF Fbs.GroupCtrlFb.Done THEN
				Fbs.GroupCtrlFb.Execute := FALSE;

				Fbs.GroupDeleteFb.Controller := ADR(gMcAcp6DController);
				Fbs.GroupDeleteFb.GroupID := 1;
				Fbs.GroupDeleteFb.Execute := TRUE;

				state := WAVE_DELETE_GROUP;
			END_IF
		WAVE_DELETE_GROUP: //**************************************************************** Delete Sh Group
			IF Fbs.GroupDeleteFb.Error THEN
				state := WAVE_ERROR;
			ELSIF Fbs.GroupDeleteFb.Done THEN
				Fbs.GroupDeleteFb.Execute := FALSE;

				Wavepars.X := 0;
				Slide.X := 0;
				state := WAVE_IDLE;
			END_IF
		WAVE_ERROR: //**************************************************************** Error State
			IF Reset THEN
				Reset := FALSE;

				Fbs.ShortAxisFb.Execute := FALSE;
				Fbs.CyclicChCtrlFb.Execute := FALSE;
				Fbs.CyclicZFb.Enable := FALSE;
				Fbs.CyclicRxFb.Enable := FALSE;
				Fbs.CyclicXFb.Enable := FALSE;
				Fbs.AutoDriveFB.Execute := FALSE;
				Fbs.GroupCreateFb.Execute := FALSE;
				Fbs.GroupCtrlFb.Execute := FALSE;
				Fbs.GroupDeleteFb.Execute := FALSE;

				Wavepars.X := 0;
				Slide.X := 0;
				state := WAVE_IDLE;
			END_IF

	END_CASE;

	Fbs.ShortAxisFb();
	Fbs.CyclicChCtrlFb();
	Fbs.CyclicZFb();
	Fbs.CyclicRxFb();
	Fbs.CyclicXFb();
	Fbs.AutoDriveFB();
	Fbs.GroupCreateFb();
	Fbs.GroupCtrlFb();
	Fbs.GroupDeleteFb();
END_PROGRAM
```

#### Init.st
```iecst
PROGRAM _INIT
	Wavepars.Center := 2.2;
	Wavepars.Amp := 1.0;
	defaultLevitationHeight := 0.001;
	shId := 1;

END_PROGRAM
```

### Program Logical/Source/Demos/AntiSlosh (IEC)

#### Types.typ
```iecst
TYPE
	AntiSloshParTyp : 	STRUCT
		ShId : USINT;
		NonSloshShId : USINT;
		ContainerLength : REAL;
		FillHeight : REAL;
		ContainerType : SFBcontShapeEnum;
		AdvPars : SFBcontAdvancedType;
		ProfilePars : MTProfilePositionParameterType;
		Payload : REAL;
		DestPos : REAL;
	END_STRUCT;
	AntiSloshIntTyp : 	STRUCT
		State : AntiSloshStatesEnum;
		ErrorState : AntiSloshStatesEnum;
		Fbs : AntiSloshFbsTyp;
		ContainerCalculated : BOOL;
	END_STRUCT;
	AntiSloshFbsTyp : 	STRUCT
		ShaperFb : SFBshaper;
		ContainerFb : SFBcontainer;
		AxisFb : MpAxisBasic;
		CylcicPosFb : MC_BR_MoveCyclicPosition;
		CyclicChCtrlFb : MC_BR_WriteCyclicChCtrl_Acp6D;
		CyclicXFb : MC_BR_WriteCyclicCh_Acp6D;
		MoveCyclicPosFb : MC_BR_MoveCyclicPosition;
		ProfGen : MTProfilePositionGenerator;
		ShPropFb : MC_BR_ShSetProperty_Acp6D;
		ShortAxisFb : MC_BR_MoveShortAxis_Acp6D;
		MovePlaneFb : MC_BR_MoveInPlane_Acp6D;
		SettleTon : TON;
	END_STRUCT;
	AntiSloshStatesEnum :
		(
		AS_IDLE,
		AS_POWER_AXIS,
		AS_HOME_AXIS,
		AS_HOME_GENERATOR,
		AS_CALC_PARS,
		AS_SET_HEIGHT,
		AS_SET_PAYLOAD,
		AS_SETUP_CYCLIC_CHANNEL,
		AS_ENABLE_CHANNEL,
		AS_SETUP_CYCLIC_AXIS_CTRL,
		AS_WAIT_MOVE,
		AS_MOVE,
		AS_DISABLE_CHANNEL,
		AS_RESET_HEIGHT,
		AS_RESET_PAYLOAD,
		AS_ERROR,
		AS_RESET
		);
END_TYPE
```

#### Variables.var
```iecst
VAR
	AxisPars : MpAxisBasicParType;
	Fbs : AntiSloshFbsTyp;
	errorState : AntiSloshStatesEnum;
	state : AntiSloshStatesEnum;
	ProfGenHomed : BOOL;
	Pars : AntiSloshParTyp;
	ContainerParsCalculated : BOOL;
	ShuttleCyclicChannelEnabled : BOOL;
	Go : BOOL;
	incAmount : REAL;
	height : REAL;
END_VAR
```

#### Cyclic.st
```iecst
PROGRAM _CYCLIC
	IF ContainerParsCalculated THEN
		Fbs.ShaperFb.In := Fbs.ProfGen.Position;
		Fbs.ShaperFb.Enable := TRUE;
	ELSE
		Fbs.ShaperFb.Enable := FALSE;
	END_IF

	IF Fbs.ShaperFb.Active AND Fbs.AxisFb.PowerOn THEN
		Fbs.MoveCyclicPosFb.Axis := ADR(gAxis_1);
		Fbs.MoveCyclicPosFb.CyclicPosition := Fbs.ShaperFb.Out;
		Fbs.MoveCyclicPosFb.Enable := TRUE;
	ELSE
		Fbs.MoveCyclicPosFb.Enable := FALSE;
	END_IF

	IF ShuttleCyclicChannelEnabled THEN
		Fbs.CyclicXFb.Value := LREAL_TO_REAL(Fbs.AxisFb.Position / 1000.0);
	END_IF

	CASE state OF
		AS_IDLE: //**************************************************************** Idle State
			IF NOT Fbs.AxisFb.PowerOn AND Fbs.AxisFb.Info.ReadyToPowerOn THEN
				Fbs.AxisFb.Power := TRUE;

				state := AS_POWER_AXIS;
			ELSIF gAntiSloshIf.Cmd.Reset THEN
				gAntiSloshIf.Cmd.Reset := FALSE;

				state := AS_RESET;
			ELSIF gAntiSloshIf.Cmd.Enable THEN
				gAntiSloshIf.Sts.Enabled := TRUE;
				Fbs.ContainerFb.Length := Pars.ContainerLength;
				Fbs.ContainerFb.FillLevel := Pars.FillHeight;
				Fbs.ContainerFb.Advanced := Pars.AdvPars;
				Fbs.ContainerFb.Shape := Pars.ContainerType;
				Fbs.ContainerFb.Enable := TRUE;

				state := AS_CALC_PARS;
			END_IF
		AS_POWER_AXIS: //**************************************************************** Power Virtual Axis
			IF Fbs.AxisFb.PowerOn THEN
				Fbs.AxisFb.Home := TRUE;

				state := AS_HOME_AXIS;
			END_IF
		AS_HOME_AXIS: //**************************************************************** Homing the virtual axis
			IF Fbs.AxisFb.Error THEN
				errorState := state;
				state := AS_ERROR;
				gAntiSloshIf.Sts.Error := TRUE;
			ELSIF Fbs.AxisFb.IsHomed AND Fbs.AxisFb.Position = AxisPars.Homing.Position THEN
				Fbs.AxisFb.Home := FALSE;

				IF NOT ProfGenHomed THEN
					Fbs.ProfGen.HomePosition := LREAL_TO_REAL(AxisPars.Homing.Position);
					Fbs.ProfGen.SetHomePosition := TRUE;
					state := AS_HOME_GENERATOR;
				ELSE
					state := AS_IDLE;
				END_IF
			END_IF
		AS_HOME_GENERATOR: //**************************************************************** Home the position generator
			IF Fbs.ProfGen.Error THEN
				errorState := state;
				state := AS_ERROR;
			ELSIF Fbs.ProfGen.Done THEN
				Fbs.ProfGen.SetHomePosition := FALSE;
				ProfGenHomed := TRUE;
				state := AS_IDLE;
			END_IF
		AS_CALC_PARS: //**************************************************************** Calculating the Anti-Slosh parameters
			IF Fbs.ContainerFb.Error THEN
				errorState := state;
				gAntiSloshIf.Sts.Error := TRUE;
				state := AS_ERROR;
			ELSIF Fbs.ContainerFb.Done THEN
				Fbs.ContainerFb.Enable := FALSE;

				ContainerParsCalculated := TRUE;
				Fbs.ShaperFb.Parameters := Fbs.ContainerFb.Result;

				Fbs.ShortAxisFb.Controller := ADR(gMcAcp6DController);
				Fbs.ShortAxisFb.ShuttleID := 1;
				Fbs.ShortAxisFb.PositionZ := height;
				Fbs.ShortAxisFb.VelocityZ := 1.0;
				Fbs.ShortAxisFb.Execute := TRUE;

				state := AS_SET_HEIGHT;

			END_IF
		AS_SET_HEIGHT: //**************************************************************** Set the shuttle's height
			IF Fbs.ShortAxisFb.Error THEN
				gAntiSloshIf.Sts.Error := TRUE;
				errorState := state;
				state := AS_ERROR;
			ELSIF Fbs.ShortAxisFb.Done THEN
				Fbs.ShortAxisFb.Execute := FALSE;

				Fbs.ShPropFb.Controller := ADR(gMcAcp6DController);
				Fbs.ShPropFb.ShuttleID[0] := Pars.ShId;
				Fbs.ShPropFb.NumberOfProperties := 1;
				Fbs.ShPropFb.Property[0] := mcACP6D_PROPERTY_PAYLOAD;
				Fbs.ShPropFb.Value[0] := Pars.Payload;
				Fbs.ShPropFb.Execute := TRUE;

				state := AS_SET_PAYLOAD;
			END_IF
		AS_SET_PAYLOAD: //**************************************************************** Set the shuttle's height
			IF Fbs.ShPropFb.Error THEN
				gAntiSloshIf.Sts.Error := TRUE;
				errorState := state;
				state := AS_ERROR;
			ELSIF Fbs.ShPropFb.Done THEN
				Fbs.ShPropFb.Execute := FALSE;
				Fbs.CyclicChCtrlFb.Controller := ADR(gMcAcp6DController);
				Fbs.CyclicChCtrlFb.ShuttleID[0] := 1;
				Fbs.CyclicChCtrlFb.ChannelID[0] := 2;
				Fbs.CyclicChCtrlFb.AxisID[0].0 := TRUE; //X
				Fbs.CyclicChCtrlFb.Execute := TRUE;
				Fbs.CyclicChCtrlFb.NumberOfShuttles := 1;
				Fbs.CyclicChCtrlFb.Level := 1;
				Fbs.CyclicChCtrlFb.OffsetX[0] := 0.060;

				state := AS_SETUP_CYCLIC_CHANNEL;
			END_IF
		AS_SETUP_CYCLIC_CHANNEL: //**************************************************************** Configuring Cyclic Channel

			IF Fbs.CyclicChCtrlFb.Error THEN
				errorState := state;
				gAntiSloshIf.Sts.Error := TRUE;
				state := AS_ERROR;
			ELSIF Fbs.CyclicChCtrlFb.Done THEN
				Fbs.CyclicChCtrlFb.Execute := FALSE;

				Fbs.CyclicXFb.Controller := ADR(gMcAcp6DController);
				Fbs.CyclicXFb.AxisID := 1;
				Fbs.CyclicXFb.ChannelID := 2;
				Fbs.CyclicXFb.Value := LREAL_TO_REAL(Fbs.AxisFb.Position / 1000.0);
				Fbs.CyclicXFb.Enable := TRUE;

				state := AS_ENABLE_CHANNEL;
			END_IF

		AS_ENABLE_CHANNEL: //**************************************************************** Starting to write to the cyclic channel
			IF Fbs.CyclicXFb.Valid THEN
				ShuttleCyclicChannelEnabled := TRUE;

				Fbs.SettleTon.PT := T#3s;
				Fbs.SettleTon.IN := TRUE;

				state := AS_WAIT_MOVE;
			END_IF
		AS_WAIT_MOVE: //**************************************************************** waiting for a move command
			IF NOT gAntiSloshIf.Cmd.Enable THEN
				Fbs.CyclicXFb.Enable := FALSE;

				Fbs.CyclicChCtrlFb.Level := 0;
				Fbs.CyclicChCtrlFb.Execute := TRUE;

				state := AS_DISABLE_CHANNEL;
			ELSIF Fbs.SettleTon.Q THEN
				Fbs.SettleTon.IN := FALSE;
				IF Fbs.ProfGen.Position = 360 THEN
					Fbs.MovePlaneFb.PositionX := 0.06;
					Pars.DestPos := 0;

				ELSE
					Fbs.MovePlaneFb.PositionX := 0.42;
					Pars.DestPos := 360;
				END_IF

				Fbs.MovePlaneFb.Controller := ADR(gMcAcp6DController);
				Fbs.MovePlaneFb.PositionY := 0.18;
				Fbs.MovePlaneFb.ShuttleID := 2;
				Fbs.MovePlaneFb.Velocity := 1;
				Fbs.MovePlaneFb.Acceleration := 10;
				Fbs.MovePlaneFb.Execute := TRUE;
				Fbs.ProfGen.Start := TRUE;

				Fbs.ProfGen.EndPosition := Pars.DestPos;
				state := AS_MOVE;
			END_IF
		AS_MOVE: //**************************************************************** Move shuttles
			IF Fbs.MovePlaneFb.Error THEN
				errorState := state;
				gAntiSloshIf.Sts.Error := TRUE;
				state := AS_ERROR;
			ELSIF gAntiSloshIf.Cmd.Reset THEN
				gAntiSloshIf.Cmd.Reset := FALSE;
				Fbs.CyclicXFb.Enable := FALSE;

				Fbs.CyclicChCtrlFb.Level := 0;
				Fbs.CyclicChCtrlFb.Execute := TRUE;
				state := AS_DISABLE_CHANNEL;
			ELSIF Fbs.MovePlaneFb.Done AND Fbs.AxisFb.Position <= Pars.DestPos + 0.1 AND Fbs.AxisFb.Position >= Pars.DestPos - 0.1 THEN
				Fbs.ProfGen.Start := FALSE;
				Fbs.MovePlaneFb.Execute := FALSE;

				Fbs.SettleTon.IN := TRUE;
				state := AS_WAIT_MOVE;
			END_IF
		AS_DISABLE_CHANNEL: //**************************************************************** Disable Channel
			IF Fbs.CyclicChCtrlFb.Error THEN
				errorState := state;
				gAntiSloshIf.Sts.Error := TRUE;
				state := AS_ERROR;
			ELSIF Fbs.CyclicChCtrlFb.Done THEN
				Fbs.CyclicChCtrlFb.Execute := FALSE;
				ShuttleCyclicChannelEnabled := FALSE;

				//Have to do this to reset the cyclic position on the 6D, for some reason otherwise it'll just error and it's really awkward to troubleshoot
				Fbs.CyclicXFb.Value := 0;
				Fbs.CyclicXFb.Enable := TRUE;

				Fbs.ShortAxisFb.PositionZ := 0.001;
				Fbs.ShortAxisFb.Execute := TRUE;

				state := AS_RESET_HEIGHT;
			END_IF
		AS_RESET_HEIGHT: //**************************************************************** Reset Shuttle Height
			IF Fbs.ShortAxisFb.Error THEN
				gAntiSloshIf.Sts.Error := TRUE;
				errorState := state;
				state := AS_ERROR;
			ELSIF Fbs.ShortAxisFb.Done THEN
				Fbs.ShortAxisFb.Execute := FALSE;
				Fbs.CyclicXFb.Enable := FALSE;

				Fbs.ShPropFb.Value[0] := 0;
				Fbs.ShPropFb.Execute := TRUE;

				state := AS_RESET_PAYLOAD;
			END_IF
		AS_RESET_PAYLOAD: //**************************************************************** Reset Payload
			IF Fbs.ShPropFb.Error THEN
				gAntiSloshIf.Sts.Error := TRUE;
				errorState := state;
				state := AS_ERROR;
			ELSIF Fbs.ShPropFb.Done THEN
				Fbs.ShPropFb.Execute := FALSE;

				state := AS_RESET;
			END_IF
		AS_ERROR: //**************************************************************** Error State
			IF gAntiSloshIf.Cmd.Reset THEN
				state := AS_RESET;
			END_IF
		AS_RESET: //**************************************************************** Reset State

			gAntiSloshIf.Sts.Enabled := FALSE;
			gAntiSloshIf.Sts.Error := FALSE;
			gAntiSloshIf.Sts.Processing := FALSE;

			gAntiSloshIf.Cmd.Reset := FALSE;

			Fbs.ContainerFb.Enable := FALSE;
			Fbs.CyclicChCtrlFb.Execute := FALSE;
			Fbs.CyclicXFb.Enable := FALSE;
			Fbs.MoveCyclicPosFb.Enable := FALSE;
			Fbs.ShaperFb.Enable := FALSE;
			Fbs.ShortAxisFb.Execute := FALSE;
			Fbs.MovePlaneFb.Execute := FALSE;
			Fbs.SettleTon.IN := FALSE;
			Fbs.ShPropFb.Execute := FALSE;

			ShuttleCyclicChannelEnabled := FALSE;
			ContainerParsCalculated := FALSE;
			ProfGenHomed := FALSE;

			Fbs.AxisFb.ErrorReset := TRUE;

			IF NOT Fbs.AxisFb.Error THEN
				Fbs.AxisFb.ErrorReset := FALSE;
				Fbs.AxisFb.Power := FALSE;

				state := AS_IDLE;
			END_IF

	END_CASE;

	Fbs.AxisFb();
	IF Fbs.AxisFb.Error AND Fbs.AxisFb.ErrorReset THEN
		Fbs.AxisFb.ErrorReset := FALSE;
		Fbs.AxisFb();
	END_IF
	Fbs.ContainerFb();
	Fbs.CyclicChCtrlFb();
	Fbs.CyclicXFb();
	Fbs.MoveCyclicPosFb();
	Fbs.ProfGen();
	Fbs.ShaperFb();
	Fbs.ShPropFb();
	Fbs.MovePlaneFb();
	Fbs.ShortAxisFb();
	Fbs.SettleTon();
END_PROGRAM
```

#### Init.st
```iecst
PROGRAM _INIT
	Fbs.AxisFb.MpLink := ADR(gAxis_1);
	Fbs.AxisFb.Parameters := ADR(AxisPars);
	Fbs.AxisFb.Enable := TRUE;
	Fbs.AxisFb();

	height := 0.001;

	Pars.ProfilePars.AccelerationNegDirection := 5000;
	Pars.ProfilePars.AccelerationPosDirection := 5000;
	Pars.ProfilePars.DecelerationNegDirection := 5000;
	Pars.ProfilePars.DecelerationPosDirection := 5000;
	Pars.ProfilePars.VelocityPosDirection := 1000;
	Pars.ProfilePars.VelocityNegDirection := 1000;

	Fbs.ProfGen.Enable := TRUE;
	Fbs.ProfGen.Parameter := Pars.ProfilePars;
	Fbs.ProfGen.HomePosition := 0;
	Fbs.ProfGen();

	Pars.ContainerLength := 0.065;
	Pars.FillHeight := 0.0325;
	AxisPars.Homing.Position := 0;

END_PROGRAM
```

### Program Logical/Source/Demos/VarDemos (IEC)

#### Cyclic.st - Cyclic code
```iecst
(*

*)

PROGRAM _CYCLIC
	IF gVariousDemoIf.Cmd.Reset THEN
		gAntiSloshIf.Cmd.Reset := TRUE;
	END_IF
	CASE state OF
		VAR_DEMO_IDLE: //******************************************************************************** Idle Wait State
			IF gVariousDemoIf.Cmd.RunDemo OR gVariousDemoIf.Cmd.ChangeDemo THEN
				gVariousDemoIf.Cmd.ChangeDemo := FALSE;
				gVariousDemoIf.Cmd.RunDemo := FALSE;

				gVariousDemoIf.Sts.Active := TRUE;
				CASE gVariousDemoIf.Par.Demo OF
					VAR_DEMO_SLIDE:
						AsignSlideDemo;
					VAR_DEMO_MIX:
						AsignMixDemo;
					VAR_DEMO_WEIGH:
						AsignWeighDemo;
					VAR_DEMO_WAVE:
						AsignWaveDemo;
					VAR_DEMO_FORCE:
						AsignForceDemo;
					VAR_DEMO_LAND:
						AsignLandDemo;
					VAR_DEMO_ANTI_SLOSH:
						AsignAntiSLosh;
					VAR_DEMO_GENERIC_MOVEMENT:
						AsignGenericDemoMovement;

				END_CASE
				Fbs.AutoDriveFb.Execute := TRUE;
				state := VAR_DEMO_MOVE_TO_START;
			END_IF
		VAR_DEMO_MOVE_TO_START: //******************************************************************************** Moving to start
			IF Fbs.AutoDriveFb.Error THEN
				state := VAR_DEMO_ERROR;
				gVariousDemoIf.Sts.Error := TRUE;
			ELSIF Fbs.AutoDriveFb.Done THEN
				Fbs.AutoDriveFb.Execute := FALSE;
				CASE gVariousDemoIf.Par.Demo OF
					VAR_DEMO_SLIDE:
						Fbs.SlideFb.Enable := TRUE;
					VAR_DEMO_MIX:
						Fbs.MixProfFb[0].Enable := TRUE;
						Fbs.MixProfFb[1].Enable := TRUE;
					VAR_DEMO_WEIGH:
//						Fbs.WeighFB[0].Execute := TRUE;
//						Fbs.WeighFB[1].Execute := TRUE;
					VAR_DEMO_WAVE:
						Fbs.WaveFb.Enable := TRUE;
					VAR_DEMO_FORCE:
						Fbs.ForceCtrlFB[0].Enable := TRUE;
						Fbs.ForceCtrlFB[1].Enable := TRUE;
					VAR_DEMO_LAND:
						Fbs.LandCtrlFb[0].Enable := TRUE;
						Fbs.LandCtrlFb[1].Enable := TRUE;
					VAR_DEMO_ANTI_SLOSH:
						gAntiSloshIf.Cmd.Enable := TRUE;
					VAR_DEMO_GENERIC_MOVEMENT:
						Fbs.GenericDemoFb.Enable := TRUE;
				END_CASE
				gVariousDemoIf.Sts.Running := TRUE;
				state := VAR_DEMO_RUN;
			END_IF
		VAR_DEMO_RUN: //******************************************************************************** Run Demo
			CASE gVariousDemoIf.Par.Demo OF
				VAR_DEMO_WEIGH:
					Fbs.WeighFB[0].Execute := NOT Fbs.WeighFB[0].Done;
					Fbs.WeighFB[1].Execute := NOT Fbs.WeighFB[1].Done;
			END_CASE

			IF Fbs.SlideFb.Error
				OR Fbs.MixProfFb[0].Error
				OR Fbs.MixProfFb[1].Error
				OR Fbs.WeighFB[0].Error
				OR Fbs.WeighFB[1].Error
				OR Fbs.WaveFb.Error
				OR Fbs.ForceCtrlFB[0].Error
				OR Fbs.ForceCtrlFB[1].Error
				OR Fbs.LandCtrlFb[0].Error
				OR Fbs.LandCtrlFb[1].Error
				OR gAntiSloshIf.Sts.Error
				OR Fbs.GenericDemoFb.Error
				THEN

				gVariousDemoIf.Sts.Error := TRUE;
				state := VAR_DEMO_ERROR;
			ELSIF gVariousDemoIf.Cmd.Stop OR gVariousDemoIf.Cmd.ChangeDemo THEN
				gVariousDemoIf.Cmd.Stop := FALSE;
				Fbs.SlideFb.Enable := FALSE;
				Fbs.MixProfFb[0].Enable := FALSE;
				Fbs.MixProfFb[1].Enable := FALSE;
				Fbs.WeighFB[0].Execute := FALSE;
				Fbs.WeighFB[1].Execute := FALSE;
				Fbs.ForceCtrlFB[0].Enable := FALSE;
				Fbs.ForceCtrlFB[1].Enable := FALSE;
				Fbs.LandCtrlFb[0].Enable := FALSE;
				Fbs.LandCtrlFb[1].Enable:= FALSE;
				Fbs.GenericDemoFb.Enable := FALSE;
				gAntiSloshIf.Cmd.Enable := FALSE;

				Fbs.WaveFb.Enable := FALSE;
				state := VAR_DEMO_STOP;
			END_IF
		VAR_DEMO_STOP: //******************************************************************************** Stopping the demo
			IF Fbs.SlideFb.Error
				OR Fbs.MixProfFb[0].Error
				OR Fbs.MixProfFb[1].Error
				OR Fbs.WaveFb.Error
				OR gAntiSloshIf.Sts.Error
				OR Fbs.GenericDemoFb.Error THEN

				gVariousDemoIf.Sts.Error := TRUE;
				state := VAR_DEMO_ERROR;
			ELSIF NOT Fbs.SlideFb.Active AND NOT Fbs.MixProfFb[0].Active
				AND NOT Fbs.MixProfFb[1].Active
				AND NOT Fbs.WeighFB[0].Active
				AND NOT Fbs.WeighFB[1].Active
				AND NOT Fbs.ForceCtrlFB[0].Active
				AND NOT Fbs.ForceCtrlFB[1].Active
				AND NOT Fbs.LandCtrlFb[0].Active
				AND NOT Fbs.LandCtrlFb[1].Active
				AND NOT gAntiSloshIf.Sts.Enabled
				AND NOT Fbs.GenericDemoFb.Active THEN

				Fbs.DelayFb.PT := delayTime;
				Fbs.DelayFb.IN := TRUE;
				IF Fbs.DelayFb.Q THEN
					Fbs.DelayFb.IN := FALSE;
					IF gVariousDemoIf.Cmd.ChangeDemo THEN
						state := VAR_DEMO_IDLE;
					ELSE
						state := VAR_DEMO_RESET;
					END_IF
				END_IF
			END_IF
		VAR_DEMO_ERROR: //******************************************************************************** Error present
			IF gVariousDemoIf.Cmd.Reset THEN
				state := VAR_DEMO_RESET;
			END_IF
		VAR_DEMO_RESET: //******************************************************************************** Resetting Everything
			gVariousDemoIf.Cmd.Reset := FALSE;

			gVariousDemoIf.Sts.Active := FALSE;
			gVariousDemoIf.Sts.Error := FALSE;
			gVariousDemoIf.Sts.Running := FALSE;
			Fbs.AutoDriveFb.Execute := FALSE;
			Fbs.MixProfFb[0].Enable := FALSE;
			Fbs.MixProfFb[1].Enable := FALSE;
			Fbs.WeighFB[0].Execute := FALSE;
			Fbs.WeighFB[1].Execute := FALSE;
			Fbs.ForceCtrlFB[0].Enable := FALSE;
			Fbs.ForceCtrlFB[1].Enable := FALSE;
			Fbs.WaveFb.Enable := FALSE;
			Fbs.LandCtrlFb[0].Enable := FALSE;
			Fbs.LandCtrlFb[1].Enable := FALSE;
			gAntiSloshIf.Cmd.Enable := FALSE;
			gAntiSloshIf.Cmd.Reset := TRUE;
			Fbs.GenericDemoFb.Enable := FALSE;
			IF NOT gAntiSloshIf.Sts.Error THEN
				state := VAR_DEMO_IDLE;
			END_IF
	END_CASE

	Fbs.AutoDriveFb();
	Fbs.SlideFb();
	Fbs.MixProfFb[0]();
	Fbs.MixProfFb[1]();
	Fbs.DelayFb();
	Fbs.WeighFB[0]();
	Fbs.WeighFB[1]();
	Fbs.ForceCtrlFB[0]();
	Fbs.ForceCtrlFB[1]();
	Fbs.LandCtrlFb[0]();
	Fbs.LandCtrlFb[1]();
	Fbs.WaveFb();
	Fbs.GenericDemoFb();

	HmiConnections;
END_PROGRAM
```

#### Init.st - Init code
```iecst
PROGRAM _INIT

	delayTime := T#400ms;

	Fbs.ForceCtrlFB[0].Controller := ADR(gMcAcp6DController);
	Fbs.ForceCtrlFB[0].Pars := ADR(forcePars[0]);

	mixPars[0].MixTime := T#4s;
	mixPars[1].MixTime := T#4s;
END_PROGRAM
```

#### Types.typ - Local data types
```iecst
TYPE
	FbsTyp : 	STRUCT
		SlideFb : SlideUpDownFb;
		MixProfFb : ARRAY[0..1]OF MixProfileFb;
		AutoDriveFb : MC_BR_MoveInPlaneAsync_Acp6D;
		DelayFb : TON;
		WeighFB : ARRAY[0..1]OF WeighShuttleFb;
		ForceCtrlFB : ARRAY[0..1]OF ForceCtrlFb;
		WaveFb : WaveFb;
		LandCtrlFb : ARRAY[0..1]OF LandFb;
		GenericDemoFb : GenericMotionDemoFB;
	END_STRUCT;
	VariousDemoStateEnum :
		(
		VAR_DEMO_IDLE,
		VAR_DEMO_MOVE_TO_START,
		VAR_DEMO_RUN,
		VAR_DEMO_STOP,
		VAR_DEMO_ERROR,
		VAR_DEMO_RESET
		);
	DemoHmiTyp : 	STRUCT
		ModeChangable : BOOL;
		ResetEnable : BOOL;
		StopEnable : BOOL;
		RunEnable : BOOL;
	END_STRUCT;
END_TYPE
```

#### Variables.var - Local variables
```iecst
VAR
	state : VariousDemoStateEnum;
	slidePars : SlideUpDownParTyp;
	mixPars : ARRAY[0..1] OF MixProfileParTyp;
	Fbs : FbsTyp;
	delayTime : TIME;
	weighPars : ARRAY[0..1] OF WeighShuttleParTyp;
	forcePars : ARRAY[0..1] OF ForceCtrlParTyp;
	wavePars : WaveParTyp;
	hmiIf : DemoHmiTyp;
	landPars : ARRAY[0..1] OF LandParsTyp;
	genDemoPars : GenDemoParType;
END_VAR
```

#### HmiConnections.st
```iecst
ACTION HmiConnections:
	hmiIf.ModeChangable := NOT gVariousDemoIf.Sts.Active AND NOT gVariousDemoIf.Sts.Running AND NOT gVariousDemoIf.Sts.Error;
	hmiIf.ResetEnable := gAntiSloshIf.Sts.Error OR gVariousDemoIf.Sts.Error;
	hmiIf.StopEnable := gVariousDemoIf.Sts.Active OR gVariousDemoIf.Sts.Running;
	hmiIf.RunEnable := NOT gVariousDemoIf.Sts.Active AND gAcp6DCtrlIf.Sts.PowerOn;
END_ACTION
```

#### AsignSlideDemo.st
```iecst
ACTION AsignSlideDemo:
	slidePars.GrpId := 1;
	slidePars.Shuttles[0].Id := 1;
	slidePars.Shuttles[0].MacroId := 135;
	slidePars.Shuttles[1].Id := 2;
	slidePars.Shuttles[1].MacroId := 136;
	slidePars.VirtualShuttle.Id := 100;
	slidePars.MoveVelocity := 1;
	slidePars.MoveDistance := 0.240;
	slidePars.MoveAcceleration := 10;
	slidePars.StartPositions[0].X := 0.060;
	slidePars.StartPositions[1].X := 0.180;
	slidePars.StartPositions[0].Y := 0.120;
	slidePars.StartPositions[1].Y := 0.120;

	Fbs.AutoDriveFb.Controller := ADR(gMcAcp6DController);
	Fbs.AutoDriveFb.NumberOfShuttles := 2;
	Fbs.AutoDriveFb.ShuttleID[0] := slidePars.Shuttles[0].Id;
	Fbs.AutoDriveFb.ShuttleID[1] := slidePars.Shuttles[1].Id;
	Fbs.AutoDriveFb.Velocity := 0.5;
	Fbs.AutoDriveFb.Acceleration := 2;
	Fbs.AutoDriveFb.PositionX[0] := slidePars.StartPositions[0].X;
	Fbs.AutoDriveFb.PositionX[1] := slidePars.StartPositions[1].X;
	Fbs.AutoDriveFb.PositionY[0] := slidePars.StartPositions[0].Y;
	Fbs.AutoDriveFb.PositionY[1] := slidePars.StartPositions[1].Y;

	Fbs.SlideFb.Controller := ADR(gMcAcp6DController);
	Fbs.SlideFb.Pars := ADR(slidePars);
	gVariousDemoIf.Sts.CurrentDemo := VAR_DEMO_SLIDE;
END_ACTION
```

#### AsignMixDemo.st
```iecst
ACTION AsignMixDemo:
	mixPars[0].VirtualShuttle.Id := 0;
	mixPars[0].VirtualShuttle.MacroId := 138;
	mixPars[0].Shuttle.Id := 1;
	mixPars[0].Shuttle.MacroId := 139;
	mixPars[0].StartPosition.X := 0.125;
	mixPars[0].StartPosition.Y := 0.125;
	mixPars[0].LevitationHeight := 0.001;

	mixPars[1].VirtualShuttle.Id := 0;
	mixPars[1].VirtualShuttle.MacroId := 138;
	mixPars[1].Shuttle.Id := 2;
	mixPars[1].Shuttle.MacroId := 138;
	mixPars[1].StartPosition.X := 0.365;
	mixPars[1].StartPosition.Y := 0.125;
	mixPars[1].LevitationHeight := 0.001;

	Fbs.MixProfFb[0].Controller := ADR(gMcAcp6DController);
	Fbs.MixProfFb[0].Pars := ADR(mixPars[0]);

	Fbs.MixProfFb[1].Controller := ADR(gMcAcp6DController);
	Fbs.MixProfFb[1].Pars := ADR(mixPars[1]);

	Fbs.AutoDriveFb.Controller := ADR(gMcAcp6DController);
	Fbs.AutoDriveFb.Velocity := 0.5;
	Fbs.AutoDriveFb.Acceleration := 2;
	Fbs.AutoDriveFb.NumberOfShuttles := 2;
	Fbs.AutoDriveFb.ShuttleID[0] := mixPars[0].Shuttle.Id;
	Fbs.AutoDriveFb.ShuttleID[1] := mixPars[1].Shuttle.Id;
	Fbs.AutoDriveFb.PositionX[0] := mixPars[0].StartPosition.X;
	Fbs.AutoDriveFb.PositionX[1] := mixPars[1].StartPosition.X;
	Fbs.AutoDriveFb.PositionY[0] := mixPars[0].StartPosition.Y;
	Fbs.AutoDriveFb.PositionY[1] := mixPars[1].StartPosition.Y;

	gVariousDemoIf.Sts.CurrentDemo := VAR_DEMO_MIX;
END_ACTION
```

#### AsignWeighDemo.st
```iecst
ACTION AsignWeighDemo:
	//weighPars[0].SettleTime := T#500ms;
	weighPars[0].ShId := 1;
	weighPars[0].TareWeight := -0.013;
	weighPars[0].StartPosition.X := 0.060;
	weighPars[0].StartPosition.Y := 0.060;

	//weighPars[1].SettleTime := T#500ms;
	weighPars[1].ShId := 2;
	weighPars[1].TareWeight := -0.0325;
	weighPars[1].StartPosition.X := 0.420;
	weighPars[1].StartPosition.Y := 0.060;

	Fbs.WeighFB[0].Controller := ADR(gMcAcp6DController);
	Fbs.WeighFB[0].Pars := ADR(weighPars[0]);

	Fbs.WeighFB[1].Controller := ADR(gMcAcp6DController);
	Fbs.WeighFB[1].Pars := ADR(weighPars[1]);

	Fbs.AutoDriveFb.Controller := ADR(gMcAcp6DController);
	Fbs.AutoDriveFb.Velocity := 0.5;
	Fbs.AutoDriveFb.Acceleration := 2;
	Fbs.AutoDriveFb.NumberOfShuttles := 2;
	Fbs.AutoDriveFb.ShuttleID[0] := weighPars[0].ShId;
	Fbs.AutoDriveFb.ShuttleID[1] := weighPars[1].ShId;
	Fbs.AutoDriveFb.PositionX[0] := weighPars[0].StartPosition.X;
	Fbs.AutoDriveFb.PositionX[1] := weighPars[1].StartPosition.X;
	Fbs.AutoDriveFb.PositionY[0] := weighPars[0].StartPosition.Y;
	Fbs.AutoDriveFb.PositionY[1] := weighPars[1].StartPosition.Y;

	gVariousDemoIf.Sts.CurrentDemo := VAR_DEMO_WEIGH;
END_ACTION
```

#### AsignWaveDemo.st
```iecst
ACTION AsignWaveDemo:
	wavePars.DefaultLevitationHeight := 0.001;

	wavePars.StartPosition[0].X := 0.420;
	wavePars.StartPosition[0].Y := 0.055;
	wavePars.StartPosition[1].X := 0.420;
	wavePars.StartPosition[1].Y := 0.185;

	wavePars.Wave.Center := 2.2;
	wavePars.Wave.Amp := 1.0;

	wavePars.Wave.Freq := 1.5;
	wavePars.Slide.Freq := 0.05;

	Fbs.WaveFb.Controller := ADR(gMcAcp6DController);
	Fbs.WaveFb.Pars := ADR(wavePars);

	Fbs.AutoDriveFb.Controller := ADR(gMcAcp6DController);
	Fbs.AutoDriveFb.Velocity := 2;
	Fbs.AutoDriveFb.Acceleration := 0.5;
	Fbs.AutoDriveFb.NumberOfShuttles := 2;
	Fbs.AutoDriveFb.ShuttleID[0] := 1;
	Fbs.AutoDriveFb.ShuttleID[1] := 2;
	Fbs.AutoDriveFb.PositionX[0] := wavePars.StartPosition[0].X;
	Fbs.AutoDriveFb.PositionX[1] := wavePars.StartPosition[1].X;
	Fbs.AutoDriveFb.PositionY[0] := wavePars.StartPosition[0].Y;
	Fbs.AutoDriveFb.PositionY[1] := wavePars.StartPosition[1].Y;

	gVariousDemoIf.Sts.CurrentDemo := VAR_DEMO_WAVE;
END_ACTION
```

#### AsignForceDemo.st
```iecst
ACTION AsignForceDemo:
	forcePars[0].ShId := 1;
	forcePars[0].ForceX := 0;
	forcePars[0].ForceY := 0;

	forcePars[0].StartPosition.X := 0.12;
	forcePars[0].StartPosition.Y := 0.12;

	forcePars[0].ForceMode := mcACP6D_FORCE_MODE_X_AXIS;

	forcePars[1].ShId := 2;
	forcePars[1].ForceX := 0;
	forcePars[1].ForceY := 0;

	forcePars[1].StartPosition.X := 0.36;
	forcePars[1].StartPosition.Y := 0.12;

	forcePars[1].ForceMode := mcACP6D_FORCE_MODE_X_AXIS;

	Fbs.ForceCtrlFB[0].Controller := ADR(gMcAcp6DController);
	Fbs.ForceCtrlFB[0].Pars := ADR(forcePars[0]);
	Fbs.ForceCtrlFB[1].Controller := ADR(gMcAcp6DController);
	Fbs.ForceCtrlFB[1].Pars := ADR(forcePars[1]);

	Fbs.AutoDriveFb.Controller := ADR(gMcAcp6DController);
	Fbs.AutoDriveFb.Velocity := 0.5;
	Fbs.AutoDriveFb.Acceleration := 2;
	Fbs.AutoDriveFb.NumberOfShuttles := 2;
	Fbs.AutoDriveFb.ShuttleID[0] := 1;
	Fbs.AutoDriveFb.ShuttleID[1] := 2;
	Fbs.AutoDriveFb.PositionX[0] := forcePars[0].StartPosition.X;
	Fbs.AutoDriveFb.PositionX[1] := forcePars[1].StartPosition.X;
	Fbs.AutoDriveFb.PositionY[0] := forcePars[0].StartPosition.Y;
	Fbs.AutoDriveFb.PositionY[1] := forcePars[1].StartPosition.Y;

	gVariousDemoIf.Sts.CurrentDemo := VAR_DEMO_FORCE;
END_ACTION
```

#### AsignLandDemo.st
```iecst
ACTION AsignLandDemo:
	landPars[0].ShId := 1;
	landPars[1].ShId := 2;

	landPars[0].StartPosition.X := 0.12;
	landPars[0].StartPosition.Y := 0.12;

	landPars[1].StartPosition.X := 0.36;
	landPars[1].StartPosition.Y := 0.12;

	Fbs.LandCtrlFb[0].Controller := ADR(gMcAcp6DController);
	Fbs.LandCtrlFb[0].Pars := ADR(landPars[0]);
	Fbs.LandCtrlFb[1].Controller := ADR(gMcAcp6DController);
	Fbs.LandCtrlFb[1].Pars := ADR(landPars[1]);

	Fbs.AutoDriveFb.Controller := ADR(gMcAcp6DController);
	Fbs.AutoDriveFb.Velocity := 0.5;
	Fbs.AutoDriveFb.Acceleration := 2;
	Fbs.AutoDriveFb.NumberOfShuttles := 2;
	Fbs.AutoDriveFb.ShuttleID[0] := 1;
	Fbs.AutoDriveFb.ShuttleID[1] := 2;
	Fbs.AutoDriveFb.PositionX[0] := landPars[0].StartPosition.X;
	Fbs.AutoDriveFb.PositionX[1] := landPars[1].StartPosition.X;
	Fbs.AutoDriveFb.PositionY[0] := landPars[0].StartPosition.Y;
	Fbs.AutoDriveFb.PositionY[1] := landPars[1].StartPosition.Y;

	gVariousDemoIf.Sts.CurrentDemo := VAR_DEMO_LAND;
END_ACTION
```

#### AsignAntiSLosh.st
```iecst
ACTION AsignAntiSLosh:

	Fbs.AutoDriveFb.Controller := ADR(gMcAcp6DController);
	Fbs.AutoDriveFb.Velocity := 0.5;
	Fbs.AutoDriveFb.Acceleration := 2;
	Fbs.AutoDriveFb.NumberOfShuttles := 2;
	Fbs.AutoDriveFb.ShuttleID[0] := 1;
	Fbs.AutoDriveFb.ShuttleID[1] := 2;
	Fbs.AutoDriveFb.PositionX[0] := 0.06;
	Fbs.AutoDriveFb.PositionX[1] := 0.06;
	Fbs.AutoDriveFb.PositionY[0] := 0.06;
	Fbs.AutoDriveFb.PositionY[1] := 0.18;

	gVariousDemoIf.Sts.CurrentDemo := VAR_DEMO_ANTI_SLOSH;
END_ACTION
```

#### AsignGenMoveDemo.st
```iecst
ACTION AsignGenericDemoMovement:
	genDemoPars.ShId[0] := 1;
	genDemoPars.ShId[1] := 2;
	genDemoPars.MacroId[0] := 140;
	genDemoPars.MacroId[1] := 141;

	genDemoPars.StartPositions[0].X := 0.240;
	genDemoPars.StartPositions[0].Y := 0.06;
	genDemoPars.StartPositions[1].X := 0.240;
	genDemoPars.StartPositions[1].Y := 0.18;

	Fbs.GenericDemoFb.Controller := ADR(gMcAcp6DController);
	Fbs.GenericDemoFb.Pars := ADR(genDemoPars);

	Fbs.AutoDriveFb.Controller := ADR(gMcAcp6DController);
	Fbs.AutoDriveFb.Velocity := 0.5;
	Fbs.AutoDriveFb.Acceleration := 2;
	Fbs.AutoDriveFb.NumberOfShuttles := 2;
	Fbs.AutoDriveFb.ShuttleID[0] := 1;
	Fbs.AutoDriveFb.ShuttleID[1] := 2;
	Fbs.AutoDriveFb.PositionX[0] := genDemoPars.StartPositions[0].X;
	Fbs.AutoDriveFb.PositionX[1] := genDemoPars.StartPositions[1].X;
	Fbs.AutoDriveFb.PositionY[0] := genDemoPars.StartPositions[0].Y;
	Fbs.AutoDriveFb.PositionY[1] := genDemoPars.StartPositions[1].Y;;

	gVariousDemoIf.Sts.CurrentDemo := VAR_DEMO_GENERIC_MOVEMENT;
END_ACTION
```

#### DemoConstants.var
```iecst
VAR CONSTANT
	rdMAX_SHUTTLE_COUNT : USINT := 2;
	rdMAX_SHUTTLE_COUNT_ARRAY : USINT := rdMAX_SHUTTLE_COUNT - 1;
END_VAR
```

#### Demos.typ
```iecst
(*Slide Up/Down Demo datatypes*)

TYPE
	SlideUpDownParTyp : 	STRUCT
		StartPositions : ARRAY[0..1]OF StationPositionTyp;
		Shuttles : ARRAY[0..1]OF ShParTyp;
		VirtualShuttle : ShParTyp;
		GrpId : USINT;
		MoveDistance : REAL;
		MoveVelocity : REAL;
		MoveAcceleration : REAL;
	END_STRUCT;
	ShParTyp : 	STRUCT
		Id : USINT;
		MacroId : USINT; (*Macro To Execute for the up/down movement*)
	END_STRUCT;
	SlideUpDownStateEnum :
		(
		SLIDE_IDLE,
		SLIDE_CREATE_GROUP,
		SLIDE_RUN_MACRO,
		SLIDE_SLIDE,
		SLIDE_STOP,
		SLIDE_DELETE_GROUP,
		SLIDE_ERROR,
		SLIDE_RESET
		);
	SlideUpDownInternalTyp : 	STRUCT
		State : SlideUpDownStateEnum;
		ErrorState : SlideUpDownStateEnum;
		Fbs : SlideUpDownFbsTyp;
	END_STRUCT;
	SlideUpDownFbsTyp : 	STRUCT
		PlanetCtrlFb : MC_BR_PlanetCtrl_Acp6D;
		RunMacroFb1 : MC_BR_MacroRun_Acp6D;
		RunMacroFb2 : MC_BR_MacroRun_Acp6D;
		MovePlaneFb : MC_BR_MoveInPlane_Acp6D;
		StopFb : MC_BR_Stop_Acp6D;
	END_STRUCT;
END_TYPE

(*Mix Profile Types*)

TYPE
	MixProfileIntTyp : 	STRUCT
		State : MixProfileStateEnum;
		ErrorState : MixProfileStateEnum;
		Fbs : MixProfileFbTyp;
	END_STRUCT;
	MixProfileParTyp : 	STRUCT
		Shuttle : ShParTyp;
		VirtualShuttle : ShParTyp;
		LevitationHeight : REAL;
		StartPosition : StationPositionTyp;
		MixTime : TIME;
	END_STRUCT;
	MixProfileFbTyp : 	STRUCT
		PlanetCtrlFb : MC_BR_PlanetCtrl_Acp6D;
		RunMacroFb : MC_BR_MacroRun_Acp6D;
		StopFb : MC_BR_Stop_Acp6D;
		MoveShortFb : MC_BR_MoveShortAxis_Acp6D;
		TimerTon : TON;
	END_STRUCT;
	MixProfileStateEnum :
		(
		MIX_IDLE,
		MIX_ENABLE_GROUP,
		MIX_RUN_MACRO_VIRT,
		MIX_RUN_MACRO_REAL,
		MIX_RUN_DEMO,
		MIX_STOP_REAL,
		MIX_STOP_VIRTUAL,
		MIX_DELETE_GROUP,
		MIX_RESET_HEIGHT,
		MIX_ERROR,
		MIX_RESET
		);
END_TYPE

(*Weight Shuttle Fb Types*)

TYPE
	WeighShuttleParTyp : 	STRUCT
		ShId : USINT;
		StartPosition : StationPositionTyp;
		TareWeight : REAL;
		SettleTime : TIME;
	END_STRUCT;
	WeighShuttleIntTyp : 	STRUCT
		State : WeighShuttleStatesEnum;
		ErrorState : WeighShuttleStatesEnum;
		Fbs : WeighShuttleFbTyp;
	END_STRUCT;
	WeighShuttleFbTyp : 	STRUCT
		SettleFb : TON;
		WeighFb : MC_BR_GetPayload_Acp6D;
	END_STRUCT;
	WeighShuttleStatesEnum :
		(
		WEIGH_IDLE,
		WEIGH_SETTLE,
		WEIGH_WEIGH,
		WEIGH_DONE,
		WEIGH_ERROR,
		WEIGH_RESET
		);
END_TYPE

(*Force Ctrl Fb Types*)

TYPE
	ForceCtrlParTyp : 	STRUCT
		ShId : USINT;
		ForceX : REAL;
		ForceY : REAL;
		ForceZ : REAL;
		ForceMode : McAcp6DForceModeLevelEnum;
		StartPosition : StationPositionTyp;
	END_STRUCT;
	ForceCtrlIntTyp : 	STRUCT
		State : ForceCtrlStatesEnum;
		ErrorState : ForceCtrlStatesEnum;
		Fbs : ForceCtrlFbsTyp;
	END_STRUCT;
	ForceCtrlFbsTyp : 	STRUCT
		ForceCtrlFb : MC_BR_ForceModeCtrl_Acp6D;
	END_STRUCT;
	ForceCtrlStatesEnum :
		(
		FORCE_IDLE,
		FORCE_ENABLE,
		FORCE_CTRL,
		FORCE_DISABLE,
		FORCE_ERROR,
		FORCE_RESET
		);
END_TYPE

(*Wave Fb Types*)

TYPE
	WaveParTyp : 	STRUCT
		Wave : SinWaveParType;
		Slide : SinWaveParType;
		DefaultLevitationHeight : REAL;
		StartPosition : ARRAY[0..1]OF StationPositionTyp;
	END_STRUCT;
	SinWaveParType : 	STRUCT
		Amp : REAL;
		Center : REAL;
		Freq : REAL;
		X : REAL;
		Y : REAL;
	END_STRUCT;
	ShuttleOutputTyp : 	STRUCT
		Height : REAL;
		Angle : REAL;
		Pos : REAL;
		WaveX : REAL;
		WaveY : REAL;
	END_STRUCT;
	WaveIntTyp : 	STRUCT
		State : WaveStateEnum;
		ErrorState : WaveStateEnum;
		WaveCtrl : ShuttleOutputTyp;
		SlideCtrl : ShuttleOutputTyp;
		Fbs : WaveFbsTyp;
	END_STRUCT;
	WaveFbsTyp : 	STRUCT
		CyclicChCtrlFb : MC_BR_WriteCyclicChCtrl_Acp6D;
		CyclicZFb : MC_BR_WriteCyclicCh_Acp6D;
		CyclicRxFb : MC_BR_WriteCyclicCh_Acp6D;
		CyclicXFb : MC_BR_WriteCyclicCh_Acp6D;
		GroupCreateFb : MC_BR_ShGroupCreate_Acp6D;
		GroupDeleteFb : MC_BR_ShGroupDelete_Acp6D;
		GroupCtrlFb : MC_BR_ShGroupCoupleCtrl_Acp6D;
		ShortAxisFb : MC_BR_MoveShortAxis_Acp6D;
	END_STRUCT;
END_TYPE

(*Anti Slosh Fb Types*)

TYPE
	WaveStateEnum :
		(
		WAVE_IDLE,
		WAVE_CREATE_GROUP,
		WAVE_BOND_GROUP,
		WAVE_CFG_CHANNEL,
		WAVE_SET_HEIGHT,
		WAVE_WAVE,
		WAVE_EXIT_CFG,
		WAVE_STOP,
		WAVE_MOVE_BACK,
		WAVE_UNBOUND_GROUP,
		WAVE_DELETE_GROUP,
		WAVE_ERROR
		);
	AntiSloshParTyp : 	STRUCT
		AxisRef : REFERENCE TO McAxisType;
		AxisPars : MpAxisBasicParType;
		ShId : USINT;
		ContainerLength : REAL;
		FillHeight : REAL;
		ContainerType : SFBcontShapeEnum;
		AdvPars : SFBcontAdvancedType;
		ProfilePars : MTProfilePositionParameterType;
	END_STRUCT;
	AntiSloshIntTyp : 	STRUCT
		State : AntiSloshStatesEnum;
		ErrorState : AntiSloshStatesEnum;
		Fbs : AntiSloshFbsTyp;
		ContainerCalculated : BOOL;
	END_STRUCT;
	AntiSloshFbsTyp : 	STRUCT
		ShaperFb : SFBshaper;
		ContainerFb : SFBcontainer;
		AxisFb : MpAxisBasic;
		CylcicPosFb : MC_BR_MoveCyclicPosition;
		CyclicChCtrlFb : MC_BR_WriteCyclicChCtrl_Acp6D;
		CyclicXFb : MC_BR_WriteCyclicCh_Acp6D;
		MoveCyclicPosFb : MC_BR_MoveCyclicPosition;
		ProfGen : MTProfilePositionGenerator;
	END_STRUCT;
	AntiSloshStatesEnum :
		(
		AS_IDLE,
		AS_ENABLE_AXIS,
		AS_POWER_AXIS,
		AS_HOME_AXIS,
		AS_CALC_PARS,
		AS_SETUP_CYCLIC_CHANNEL,
		AS_ENABLE_CHANNEL,
		AS_SETUP_CYCLIC_AXIS_CTRL,
		AS_WAIT_MOVE,
		AS_MOVE,
		AS_ERROR,
		AS_RESET
		);
END_TYPE

(*Land/Levitate Types*)

TYPE
	LandParsTyp : 	STRUCT
		ShId : USINT;
		StartPosition : StationPositionTyp;
		Move : McAcp6DLevitationLevelEnum;
	END_STRUCT;
	LandIntTyp : 	STRUCT
		State : LandStateEnum;
		ErrorState : LandStateEnum;
		Landed : BOOL;
		Fbs : LandFbsTyp;
	END_STRUCT;
	LandFbsTyp : 	STRUCT
		LandFb : MC_BR_LevitationCtrl_Acp6D;
	END_STRUCT;
	LandStateEnum :
		(
		LAND_IDLE,
		LAND_ISSUE_CMD,
		LAND_WAIT,
		LAND_ERROR,
		LAND_RESET
		);
END_TYPE

(*Generic Motion Profile Demo Types*)

TYPE
	GenDemoParType : 	STRUCT
		ShId : ARRAY[0..1]OF USINT;
		MacroId : ARRAY[0..1]OF USINT;
		StartPositions : ARRAY[0..1]OF StationPositionTyp;
	END_STRUCT;
	GenDemoStateEnum :
		(
		GEN_IDLE,
		GEN_BLOCK_BUFFER,
		GEN_RUN_MACRO1,
		GEN_RUN_MACRO2,
		GEN_RELEASE_BUFFER,
		GEN_RUN_DEMO,
		GEN_STOP,
		GEN_RESET_HEIGHT1,
		GEN_RESET_HEIGHT2,
		GEN_ERROR,
		GEN_RESET
		);
	GenDemoFbsTyp : 	STRUCT
		ShortAxisFb : MC_BR_MoveShortAxis_Acp6D;
		MacroRunFB : MC_BR_MacroRun_Acp6D;
		BufferCtrl : MC_BR_BufferCtrl_Acp6D;
		StopFb : MC_BR_Stop_Acp6D;
	END_STRUCT;
	GenDemoIntTyp : 	STRUCT
		State : GenDemoStateEnum;
		ErrorState : GenDemoStateEnum;
		Fbs : GenDemoFbsTyp;
	END_STRUCT;
END_TYPE
```

#### LocalFunctions.fun
```iecst
{REDUND_ERROR} {REDUND_UNREPLICABLE} FUNCTION_BLOCK SlideUpDownFb (*TODO: Add your comment here*) (*$GROUP=User,$CAT=User,$GROUPICON=User.png,$CATICON=User.png*)
	VAR_INPUT
		Controller : REFERENCE TO McAcp6DControllerType;
		Enable : {REDUND_UNREPLICABLE} BOOL;
		Pars : REFERENCE TO SlideUpDownParTyp;
	END_VAR
	VAR_OUTPUT
		Error : {REDUND_UNREPLICABLE} BOOL;
		Active : {REDUND_UNREPLICABLE} BOOL;
	END_VAR
	VAR
		int : {REDUND_UNREPLICABLE} SlideUpDownInternalTyp;
	END_VAR
END_FUNCTION_BLOCK

FUNCTION_BLOCK MixProfileFb
	VAR_INPUT
		Controller : REFERENCE TO McAcp6DControllerType;
		Enable : BOOL;
		Pars : REFERENCE TO MixProfileParTyp;
	END_VAR
	VAR_OUTPUT
		Error : BOOL;
		Active : BOOL;
	END_VAR
	VAR
		int : MixProfileIntTyp;
	END_VAR
END_FUNCTION_BLOCK

FUNCTION_BLOCK WeighShuttleFb
	VAR_INPUT
		Controller : REFERENCE TO McAcp6DControllerType;
		Execute : BOOL;
		Pars : REFERENCE TO WeighShuttleParTyp;
	END_VAR
	VAR_OUTPUT
		Error : BOOL;
		Active : BOOL;
		Done : BOOL;
		Weight : REAL;
	END_VAR
	VAR
		int : WeighShuttleIntTyp;
	END_VAR
END_FUNCTION_BLOCK

FUNCTION_BLOCK ForceCtrlFb
	VAR_INPUT
		Controller : REFERENCE TO McAcp6DControllerType;
		Enable : BOOL;
		Update : BOOL;
		Pars : REFERENCE TO ForceCtrlParTyp;
	END_VAR
	VAR_OUTPUT
		Error : BOOL;
		Active : BOOL;
	END_VAR
	VAR
		int : ForceCtrlIntTyp;
	END_VAR
END_FUNCTION_BLOCK

{REDUND_ERROR} FUNCTION_BLOCK WaveFb (*TODO: Add your comment here*) (*$GROUP=User,$CAT=User,$GROUPICON=User.png,$CATICON=User.png*)
	VAR_INPUT
		Controller : REFERENCE TO McAcp6DControllerType;
		Enable : {REDUND_UNREPLICABLE} BOOL;
		Pars : REFERENCE TO WaveParTyp;
	END_VAR
	VAR_OUTPUT
		Error : {REDUND_UNREPLICABLE} BOOL;
		Active : {REDUND_UNREPLICABLE} BOOL;
		Running : BOOL;
	END_VAR
	VAR
		int : {REDUND_UNREPLICABLE} WaveIntTyp;
	END_VAR
END_FUNCTION_BLOCK

{REDUND_ERROR} FUNCTION_BLOCK AntiSloshFb (*TODO: Add your comment here*) (*$GROUP=User,$CAT=User,$GROUPICON=User.png,$CATICON=User.png*)
	VAR_INPUT
		Controller : REFERENCE TO McAcp6DControllerType;
		Enable : {REDUND_UNREPLICABLE} BOOL;
		ReCalcContainer : BOOL;
		Pars : REFERENCE TO AntiSloshParTyp;
	END_VAR
	VAR_OUTPUT
		Error : {REDUND_UNREPLICABLE} BOOL;
		ContainerParsCalculated : BOOL;
		Active : {REDUND_UNREPLICABLE} BOOL;
		ShuttleWriteValid : BOOL;
		ShapeActive : BOOL;
		VirtualCyclicActive : BOOL;
	END_VAR
	VAR
		int : {REDUND_UNREPLICABLE} AntiSloshIntTyp;
	END_VAR
END_FUNCTION_BLOCK

{REDUND_ERROR} {REDUND_UNREPLICABLE} FUNCTION_BLOCK LandFb (*TODO: Add your comment here*) (*$GROUP=User,$CAT=User,$GROUPICON=User.png,$CATICON=User.png*)
	VAR_INPUT
		Controller : REFERENCE TO McAcp6DControllerType;
		Enable : {REDUND_UNREPLICABLE} BOOL;
		Land : {REDUND_UNREPLICABLE} BOOL;
		Pars : REFERENCE TO LandParsTyp;
	END_VAR
	VAR_OUTPUT
		Error : {REDUND_UNREPLICABLE} BOOL;
		Active : {REDUND_UNREPLICABLE} BOOL;
	END_VAR
	VAR
		int : {REDUND_UNREPLICABLE} LandIntTyp;
	END_VAR
END_FUNCTION_BLOCK

{REDUND_ERROR} {REDUND_UNREPLICABLE} FUNCTION_BLOCK GenericMotionDemoFB (*TODO: Add your comment here*) (*$GROUP=User,$CAT=User,$GROUPICON=User.png,$CATICON=User.png*)
	VAR_INPUT
		Controller : REFERENCE TO McAcp6DControllerType;
		Enable : {REDUND_UNREPLICABLE} BOOL;
		Land : {REDUND_UNREPLICABLE} BOOL;
		Pars : REFERENCE TO GenDemoParType;
	END_VAR
	VAR_OUTPUT
		Error : {REDUND_UNREPLICABLE} BOOL;
		Active : {REDUND_UNREPLICABLE} BOOL;
	END_VAR
	VAR
		int : {REDUND_UNREPLICABLE} GenDemoIntTyp;
	END_VAR
END_FUNCTION_BLOCK
```

#### SlideUpDownFb.st
```iecst
(* Demo implementation TO showcase robot tracking a master shuttle *)
(*
	Change robot program and call Sync Program (robot should be powered and ready to run)
	Cfg Cyclic Channel for shuttle
	Setup Sun/Planet for virtual shuttle/real shuttle
	Once ready to sync, enable online path influencer
	call loop macro on shuttle
	When no enable, stop shuttle, stop robot
	Reset

*)
FUNCTION_BLOCK SlideUpDownFb
	CASE int.State OF
		SLIDE_IDLE: //******************************************************************************** Idle Wait State
			IF Enable THEN
				int.Fbs.PlanetCtrlFb.Controller := ADR(Controller);
				int.Fbs.PlanetCtrlFb.Level := mcACP6D_PLANET_CONNECT;
				int.Fbs.PlanetCtrlFb.NumberOfPlanets := 2;
				int.Fbs.PlanetCtrlFb.StarShuttleID := Pars.VirtualShuttle.Id;
				int.Fbs.PlanetCtrlFb.PlanetShuttleID[0] := Pars.Shuttles[0].Id;
				int.Fbs.PlanetCtrlFb.PlanetShuttleID[1] := Pars.Shuttles[1].Id;
				int.Fbs.PlanetCtrlFb.Execute := TRUE;

				int.State := SLIDE_CREATE_GROUP;
			END_IF
		SLIDE_CREATE_GROUP: //******************************************************************************** Setting up the groups
			IF int.Fbs.PlanetCtrlFb.Error THEN
				int.ErrorState := int.State;
				Error := TRUE;
				int.State := SLIDE_ERROR;
			ELSIF int.Fbs.PlanetCtrlFb.Done THEN
				int.Fbs.PlanetCtrlFb.Execute := FALSE;

				int.Fbs.RunMacroFb1.Controller := ADR(Controller);
				int.Fbs.RunMacroFb1.ShuttleID := Pars.Shuttles[0].Id;
				int.Fbs.RunMacroFb1.MacroID := Pars.Shuttles[0].MacroId;
				int.Fbs.RunMacroFb1.Execute := TRUE;

				int.Fbs.RunMacroFb2.Controller := ADR(Controller);
				int.Fbs.RunMacroFb2.ShuttleID := Pars.Shuttles[1].Id;
				int.Fbs.RunMacroFb2.MacroID := Pars.Shuttles[1].MacroId;
				int.Fbs.RunMacroFb2.Execute := TRUE;

				int.State := SLIDE_RUN_MACRO;
			END_IF
		SLIDE_RUN_MACRO: //******************************************************************************** Running Macro State
			IF int.Fbs.RunMacroFb2.Error OR int.Fbs.RunMacroFb1.Error THEN
				int.ErrorState := int.State;
				Error := TRUE;
				int.State := SLIDE_ERROR;
			ELSIF int.Fbs.RunMacroFb2.Acknowledge AND int.Fbs.RunMacroFb1.Acknowledge THEN
				int.Fbs.RunMacroFb2.Execute := FALSE;
				int.Fbs.RunMacroFb1.Execute := FALSE;

				int.Fbs.MovePlaneFb.Controller := ADR(Controller);
				int.Fbs.MovePlaneFb.ShuttleID := Pars.VirtualShuttle.Id;
				int.Fbs.MovePlaneFb.Mode := mcACP6D_MOVE_RELATIVE;
				int.Fbs.MovePlaneFb.Path := mcACP6D_PATH_DIRECT;
				int.Fbs.MovePlaneFb.PositionX := Pars.MoveDistance;
				int.Fbs.MovePlaneFb.PositionY := 0;
				int.Fbs.MovePlaneFb.Velocity := Pars.MoveVelocity;
				int.Fbs.MovePlaneFb.Acceleration := Pars.MoveAcceleration;
				int.Fbs.MovePlaneFb.Execute := TRUE;

				int.State := SLIDE_SLIDE;
			END_IF
		SLIDE_SLIDE: //******************************************************************************** Slide demo state
			int.Fbs.MovePlaneFb.Execute := TRUE;
			IF int.Fbs.MovePlaneFb.Error THEN
				int.ErrorState := int.State ;
				Error := TRUE;
				int.State := SLIDE_ERROR;
			ELSIF NOT Enable THEN
				int.Fbs.MovePlaneFb.Execute := FALSE;

				int.Fbs.StopFb.Controller := ADR(Controller);
				int.Fbs.StopFb.ShuttleID := 0;
				int.Fbs.StopFb.Execute := TRUE;

				int.State := SLIDE_STOP;
			ELSIF int.Fbs.MovePlaneFb.Done THEN
				int.Fbs.MovePlaneFb.Execute := FALSE;
				int.Fbs.MovePlaneFb.PositionX := int.Fbs.MovePlaneFb.PositionX * -1; //Invert the position to move left/right

			END_IF
		SLIDE_STOP: //******************************************************************************** Stopping state
			IF int.Fbs.StopFb.Error THEN
				int.ErrorState := int.State;
				Error := TRUE;
				int.State := SLIDE_ERROR;
			ELSIF int.Fbs.StopFb.Done THEN
				int.Fbs.StopFb.Execute := FALSE;

				int.Fbs.PlanetCtrlFb.Level := mcACP6D_PLANET_DISCONNECT;
				int.Fbs.PlanetCtrlFb.Execute := TRUE;

				int.State := SLIDE_DELETE_GROUP;
			END_IF
		SLIDE_DELETE_GROUP: //******************************************************************************** Deleting the group
			IF int.Fbs.PlanetCtrlFb.Error THEN
				int.ErrorState := int.State;
				Error := TRUE;
				int.State := SLIDE_ERROR;
			ELSIF int.Fbs.PlanetCtrlFb.Done THEN
				int.Fbs.PlanetCtrlFb.Execute := FALSE;

				Active := FALSE;

				int.State := SLIDE_RESET;
			END_IF
		SLIDE_ERROR: //******************************************************************************** Error State
			IF NOT Enable THEN
				int.State := SLIDE_RESET;
			END_IF
		SLIDE_RESET: //******************************************************************************** Reset State
			Active := FALSE;
			Error := FALSE;

			int.Fbs.PlanetCtrlFb.Execute := FALSE;
			int.Fbs.MovePlaneFb.Execute := FALSE;
			int.Fbs.RunMacroFb1.Execute := FALSE;
			int.Fbs.RunMacroFb2.Execute := FALSE;
			int.Fbs.StopFb.Execute := FALSE;

			int.State := SLIDE_IDLE;

	END_CASE;

	//Call the FBs
	int.Fbs.PlanetCtrlFb();
	int.Fbs.MovePlaneFb();
	int.Fbs.RunMacroFb1();
	int.Fbs.RunMacroFb2();
	int.Fbs.StopFb();

END_FUNCTION_BLOCK
```

#### MixProfileFb.st
```iecst
(*
*)
FUNCTION_BLOCK MixProfileFb
	CASE int.State OF
		MIX_IDLE: //******************************************************************************** Idle Wait State
			IF Enable THEN
				IF Pars.VirtualShuttle.Id <> 0 THEN
					int.Fbs.PlanetCtrlFb.Controller := ADR(Controller);
					int.Fbs.PlanetCtrlFb.Level := mcACP6D_PLANET_CONNECT;
					int.Fbs.PlanetCtrlFb.StarShuttleID:= Pars.VirtualShuttle.Id;
					int.Fbs.PlanetCtrlFb.NumberOfPlanets := 1;
					int.Fbs.PlanetCtrlFb.PlanetShuttleID[0] := Pars.Shuttle.Id;
					int.Fbs.PlanetCtrlFb.Execute := TRUE;

					int.State := MIX_ENABLE_GROUP;
				ELSE
					int.Fbs.RunMacroFb.Controller := ADR(Controller);
					int.Fbs.RunMacroFb.MacroID := Pars.Shuttle.MacroId;
					int.Fbs.RunMacroFb.ShuttleID := Pars.Shuttle.Id;
					int.Fbs.RunMacroFb.Execute := TRUE;

					int.State := MIX_RUN_MACRO_REAL;
				END_IF
			END_IF
		MIX_ENABLE_GROUP:  //******************************************************************************** Enable group
			IF int.Fbs.PlanetCtrlFb.Error THEN
				int.ErrorState := int.State;
				int.State := MIX_ERROR;
			ELSIF int.Fbs.PlanetCtrlFb.Done THEN
				int.Fbs.PlanetCtrlFb.Execute := FALSE;

				int.Fbs.RunMacroFb.Controller := ADR(Controller);
				int.Fbs.RunMacroFb.MacroID := Pars.VirtualShuttle.MacroId;
				int.Fbs.RunMacroFb.ShuttleID := Pars.VirtualShuttle.Id;
				int.Fbs.RunMacroFb.Execute := TRUE;

				int.State := MIX_RUN_MACRO_VIRT;
			END_IF
		MIX_RUN_MACRO_VIRT://******************************************************************************** Run macro on virtual shuttle
			IF int.Fbs.RunMacroFb.Error THEN
				int.ErrorState := int.State;
				int.State := MIX_ERROR;
			ELSIF int.Fbs.RunMacroFb.Acknowledge THEN
				int.Fbs.RunMacroFb.Execute := FALSE;

				int.Fbs.RunMacroFb.MacroID := Pars.Shuttle.MacroId;
				int.Fbs.RunMacroFb.ShuttleID := Pars.Shuttle.Id;

				int.State := MIX_RUN_MACRO_REAL;
			END_IF
		MIX_RUN_MACRO_REAL: //******************************************************************************** RUn Maro on real shuttle
			int.Fbs.RunMacroFb.Execute := TRUE;
			IF int.Fbs.RunMacroFb.Error THEN
				int.ErrorState := int.State;
				int.State := MIX_ERROR;
			ELSIF int.Fbs.RunMacroFb.Acknowledge THEN
				int.Fbs.RunMacroFb.Execute := FALSE;

				int.Fbs.TimerTon.IN := TRUE;
				int.Fbs.TimerTon.PT := Pars.MixTime;

				int.State := MIX_RUN_DEMO;
			END_IF
		MIX_RUN_DEMO: //******************************************************************************** Running the demo
			IF NOT Enable OR int.Fbs.TimerTon.Q THEN
				int.Fbs.TimerTon.IN := FALSE;
				int.Fbs.StopFb.Controller := ADR(Controller);
				int.Fbs.StopFb.ShuttleID := Pars.VirtualShuttle.Id;
				int.Fbs.StopFb.Execute := TRUE;

				int.State := MIX_STOP_VIRTUAL;
			END_IF
		MIX_STOP_VIRTUAL: //******************************************************************************** Stopping the real shuttle
			IF int.Fbs.StopFb.Error THEN
				int.ErrorState := int.State;
				int.State := MIX_ERROR;
			ELSIF int.Fbs.StopFb.Done THEN
				int.Fbs.StopFb.Execute := FALSE;

				int.Fbs.StopFb.ShuttleID := Pars.Shuttle.Id;
				int.State := MIX_STOP_REAL;
			END_IF
		MIX_STOP_REAL: //******************************************************************************** Stopping the virtual shuttle
			int.Fbs.StopFb.Execute := TRUE;
			IF int.Fbs.StopFb.Error THEN
				int.ErrorState := int.State;
				int.State := MIX_ERROR;
			ELSIF int.Fbs.StopFb.Done THEN
				int.Fbs.StopFb.Execute := FALSE;

				IF Pars.VirtualShuttle.Id <> 0 THEN
					int.Fbs.PlanetCtrlFb.Level := mcACP6D_PLANET_DISCONNECT;
					int.Fbs.PlanetCtrlFb.Execute := TRUE;
					int.State := MIX_DELETE_GROUP;
				ELSE
					int.Fbs.MoveShortFb.Controller := ADR(Controller);
					int.Fbs.MoveShortFb.ShuttleID := Pars.Shuttle.Id;
					int.Fbs.MoveShortFb.PositionRx := 0;
					int.Fbs.MoveShortFb.PositionRy := 0;
					int.Fbs.MoveShortFb.PositionRz := 0;
					int.Fbs.MoveShortFb.PositionZ := Pars.LevitationHeight;
					int.Fbs.MoveShortFb.VelocityRx := 0.5;
					int.Fbs.MoveShortFb.VelocityRy := 0.5;
					int.Fbs.MoveShortFb.VelocityRz := 0.5;
					int.Fbs.MoveShortFb.VelocityZ := 1;
					int.Fbs.MoveShortFb.Execute := TRUE;

					int.State := MIX_RESET_HEIGHT;
				END_IF

			END_IF
		MIX_DELETE_GROUP: //******************************************************************************** Deleteing the sun/planet
			IF int.Fbs.PlanetCtrlFb.Error THEN
				int.ErrorState := int.State;
				int.State := MIX_ERROR;
			ELSIF int.Fbs.PlanetCtrlFb.Done THEN
				int.Fbs.PlanetCtrlFb.Execute := FALSE;

				int.Fbs.MoveShortFb.Controller := ADR(Controller);
				int.Fbs.MoveShortFb.ShuttleID := Pars.Shuttle.Id;
				int.Fbs.MoveShortFb.PositionRx := 0;
				int.Fbs.MoveShortFb.PositionRy := 0;
				int.Fbs.MoveShortFb.PositionRz := 0;
				int.Fbs.MoveShortFb.PositionZ := Pars.LevitationHeight;
				int.Fbs.MoveShortFb.VelocityRx := 0.5;
				int.Fbs.MoveShortFb.VelocityRy := 0.5;
				int.Fbs.MoveShortFb.VelocityRz := 0.5;
				int.Fbs.MoveShortFb.VelocityZ := 1;
				int.Fbs.MoveShortFb.Execute := TRUE;

				int.State := MIX_RESET_HEIGHT;
			END_IF
		MIX_RESET_HEIGHT: //******************************************************************************** Reset the shuttle's height
			IF int.Fbs.MoveShortFb.Error THEN
				int.ErrorState := int.State;
				int.State := MIX_ERROR;
			ELSIF int.Fbs.MoveShortFb.Done THEN
				int.Fbs.MoveShortFb.Execute := FALSE;

				Active := FALSE;
				int.State := MIX_RESET;
			END_IF
		MIX_ERROR: //******************************************************************************** Error State
			IF NOT Enable THEN
				int.State := MIX_RESET;

			END_IF
		MIX_RESET: //******************************************************************************** Reset the fbs and outputs
			Active := FALSE;
			Error := FALSE;

			int.Fbs.TimerTon.IN := FALSE;
			int.Fbs.MoveShortFb.Execute := FALSE;
			int.Fbs.PlanetCtrlFb.Execute := FALSE;
			int.Fbs.RunMacroFb.Execute := FALSE;
			int.Fbs.StopFb.Execute := FALSE;

			int.State := MIX_IDLE;
	END_CASE;

	//Call the FBs

	int.Fbs.RunMacroFb();
	//int.Fbs.TimerTon();
	int.Fbs.PlanetCtrlFb();
	int.Fbs.MoveShortFb();
	int.Fbs.StopFb();

END_FUNCTION_BLOCK
```

#### WeighShuttleFb.st
```iecst
(*
*)
FUNCTION_BLOCK WeighShuttleFb
	CASE int.State OF
		WEIGH_IDLE: //******************************************************************************** Idle Wait State
			IF Execute THEN
				Active := TRUE;

				int.Fbs.SettleFb.IN := TRUE;
				int.Fbs.SettleFb.PT := Pars.SettleTime;

				int.State := WEIGH_SETTLE;
			END_IF
		WEIGH_SETTLE:  //******************************************************************************** Waiting for settle
			IF int.Fbs.SettleFb.Q THEN
				int.Fbs.SettleFb.IN := FALSE;

				int.Fbs.WeighFb.Controller := ADR(Controller);
				int.Fbs.WeighFb.ShuttleID := Pars.ShId;
				int.Fbs.WeighFb.Execute := TRUE;

				int.State := WEIGH_WEIGH;
			END_IF
		WEIGH_WEIGH://******************************************************************************** Weighing shuttle payload
			IF int.Fbs.WeighFb.Error THEN
				int.ErrorState := int.State;
				int.State := WEIGH_ERROR;
			ELSIF int.Fbs.WeighFb.Valid THEN
				Weight := int.Fbs.WeighFb.Payload - Pars.TareWeight;
				Done := TRUE;

				int.State := WEIGH_DONE;
			END_IF
		WEIGH_DONE: //******************************************************************************** Done
			IF NOT Execute THEN
				int.State := WEIGH_RESET;
			END_IF
		WEIGH_ERROR: //******************************************************************************** Error present
			IF NOT Execute THEN
				int.State := WEIGH_RESET;
			END_IF
		WEIGH_RESET: //******************************************************************************** Reset State
			Active := FALSE;
			Done := FALSE;
			Error := FALSE;

			int.Fbs.SettleFb.IN := FALSE;
			int.Fbs.WeighFb.Execute := FALSE;

			int.State := WEIGH_IDLE;
	END_CASE;

	//Call the FBs
	int.Fbs.SettleFb();
	int.Fbs.WeighFb();

END_FUNCTION_BLOCK
```

#### ForceCtrlFb.st
```iecst
(*
*)
FUNCTION_BLOCK ForceCtrlFb
	CASE int.State OF
		FORCE_IDLE: //******************************************************************************** Idle Wait State
			IF Enable THEN
				Active := TRUE;
				Update := FALSE;

				int.Fbs.ForceCtrlFb.Controller := ADR(Controller);
				int.Fbs.ForceCtrlFb.Mode := Pars.ForceMode;
				int.Fbs.ForceCtrlFb.ForceX := Pars.ForceX;
				int.Fbs.ForceCtrlFb.ForceY := Pars.ForceY;
				int.Fbs.ForceCtrlFb.ForceZ := Pars.ForceZ;
				int.Fbs.ForceCtrlFb.ShuttleID := Pars.ShId;
				int.Fbs.ForceCtrlFb.Execute := TRUE;

				int.State := FORCE_ENABLE;
			END_IF
		FORCE_ENABLE:  //******************************************************************************** Enabling Force Ctrl
			IF int.Fbs.ForceCtrlFb.Error THEN
				int.ErrorState := int.State;
				int.State := FORCE_ERROR;
			ELSIF int.Fbs.ForceCtrlFb.Done THEN
				int.Fbs.ForceCtrlFb.Execute := FALSE;

				int.State := FORCE_CTRL;
			END_IF

		FORCE_CTRL://******************************************************************************** Force Ctrl Active
			IF NOT Enable OR Update THEN
				int.Fbs.ForceCtrlFb.Mode := mcACP6D_FORCE_MODE_EXIT;
				int.Fbs.ForceCtrlFb.Execute := TRUE;

				int.State := FORCE_DISABLE;
			END_IF
		FORCE_DISABLE: //******************************************************************************** Exiting Force Ctrl
			IF int.Fbs.ForceCtrlFb.Error THEN
				int.ErrorState := int.State;
				int.State := FORCE_ERROR;
			ELSIF int.Fbs.ForceCtrlFb.Done THEN
				int.Fbs.ForceCtrlFb.Execute := FALSE;

				IF Update THEN
					Update := FALSE;
					int.Fbs.ForceCtrlFb.Mode := Pars.ForceMode;
					int.Fbs.ForceCtrlFb.ForceX := Pars.ForceX;
					int.Fbs.ForceCtrlFb.ForceY := Pars.ForceY;
					int.Fbs.ForceCtrlFb.ForceZ := Pars.ForceZ;
					int.Fbs.ForceCtrlFb.ShuttleID := Pars.ShId;
					int.Fbs.ForceCtrlFb.Execute := TRUE;
				ELSE
					int.State := FORCE_RESET;
				END_IF

			END_IF
		FORCE_ERROR: //******************************************************************************** Error present
			IF NOT Enable THEN
				int.State := FORCE_RESET;
			END_IF
		FORCE_RESET: //******************************************************************************** Reset State
			Active := FALSE;
			Error := FALSE;

			int.Fbs.ForceCtrlFb.Execute := FALSE;

			int.State := FORCE_IDLE;
	END_CASE;

	//Call the FBs
	int.Fbs.ForceCtrlFb();

END_FUNCTION_BLOCK
```
